LIN {X 0,Y 574.087,Z 352.568,A -85,B 0,C 180,E1 -2236.257,E2 -2236.257} C_VEL
LIN {X 0,Y 573.893,Z 454.984,A -85,B 0,C 180,E1 -2237.558,E2 -2237.558} C_VEL
LIN {X 0,Y 573.782,Z 468.244,A -85,B 0,C 180,E1 -2237.87,E2 -2237.87} C_VEL
LIN {X 0,Y 573.666,Z 481.513,A -85,B 0,C 180,E1 -2238.339,E2 -2238.339} C_VEL
LIN {X 0,Y 573.595,Z 492.64,A -85,B 0,C 180,E1 -2238.874,E2 -2238.874} C_VEL
LIN {X 0,Y 573.43,Z 504.211,A -85,B 0,C 180,E1 -2239.586,E2 -2239.586} C_VEL
LIN {X 0,Y 573.326,Z 514.578,A -85,B 0,C 180,E1 -2240.386,E2 -2240.386} C_VEL
LIN {X 0,Y 573.238,Z 523.076,A -85,B 0,C 180,E1 -2241.185,E2 -2241.185} C_VEL
LIN {X 0,Y 573.16,Z 530.966,A -85,B 0,C 180,E1 -2242.072,E2 -2242.072} C_VEL
LIN {X 0,Y 573.078,Z 538.898,A -85,B 0,C 180,E1 -2243.177,E2 -2243.177} C_VEL
LIN {X 0,Y 573.07,Z 545.683,A -85,B 0,C 180,E1 -2244.37,E2 -2244.37} C_VEL
LIN {X 0,Y 573.028,Z 550.375,A -85,B 0,C 180,E1 -2245.428,E2 -2245.428} C_VEL
LIN {X 0,Y 573.023,Z 553.959,A -85,B 0,C 180,E1 -2246.485,E2 -2246.485} C_VEL
LIN {X 0,Y 572.959,Z 555.81,A -85,B 0,C 180,E1 -2247.188,E2 -2247.188} C_VEL
LIN {X 0,Y 572.946,Z 558.186,A -85,B 0,C 180,E1 -2248.595,E2 -2248.595} C_VEL
LIN {X 0,Y 572.938,Z 559,A -85,B 0,C 180,E1 -2250.001,E2 -2250.001} C_VEL
LIN {X 0,Y 572.946,Z 558.186,A -85,B 0,C 180,E1 -2251.406,E2 -2251.406} C_VEL
LIN {X 0,Y 572.937,Z 557.198,A -85,B 0,C 180,E1 -2252.11,E2 -2252.11} C_VEL
LIN {X 0,Y 572.959,Z 555.808,A -85,B 0,C 180,E1 -2252.813,E2 -2252.813} C_VEL
LIN {X 0,Y 573.014,Z 552.894,A -85,B 0,C 180,E1 -2253.869,E2 -2253.869} C_VEL
LIN {X 0,Y 572.963,Z 548.946,A -85,B 0,C 180,E1 -2254.926,E2 -2254.926} C_VEL
LIN {X 0,Y 573.067,Z 542.873,A -85,B 0,C 180,E1 -2256.161,E2 -2256.161} C_VEL
LIN {X 0,Y 573.12,Z 536.233,A -85,B 0,C 180,E1 -2257.221,E2 -2257.221} C_VEL
LIN {X 0,Y 573.192,Z 527.986,A -85,B 0,C 180,E1 -2258.284,E2 -2258.284} C_VEL
LIN {X 0,Y 573.312,Z 517.586,A -85,B 0,C 180,E1 -2259.348,E2 -2259.348} C_VEL
LIN {X 0,Y 573.427,Z 507.917,A -85,B 0,C 180,E1 -2260.148,E2 -2260.148} C_VEL
LIN {X 0,Y 573.552,Z 497.347,A -85,B 0,C 180,E1 -2260.858,E2 -2260.858} C_VEL
LIN {X 0,Y 573.654,Z 486.27,A -85,B 0,C 180,E1 -2261.448,E2 -2261.448} C_VEL
LIN {X 0,Y 573.76,Z 473.155,A -85,B 0,C 180,E1 -2261.975,E2 -2261.975} C_VEL
LIN {X 0,Y 573.831,Z 460.495,A -85,B 0,C 180,E1 -2262.332,E2 -2262.332} C_VEL
LIN {X 0,Y 573.897,Z 447.265,A -85,B 0,C 180,E1 -2262.555,E2 -2262.555} C_VEL
LIN {X 0,Y 573.953,Z 350.676,A -85,B 0,C 180,E1 -2263.77,E2 -2263.77} C_VEL
LIN {X 0,Y 573.386,Z 346.788,A -85,B 0,C 180,E1 -2263.851,E2 -2263.851} C_VEL
LIN {X 0,Y 573.57,Z 325.022,A -85,B 0,C 180,E1 -2266.994,E2 -2266.994} C_VEL
LIN {X 0,Y 573.803,Z 304.129,A -85,B 0,C 180,E1 -2270.057,E2 -2270.057} C_VEL
LIN {X 0,Y 573.969,Z 288.92,A -85,B 0,C 180,E1 -2272.308,E2 -2272.308} C_VEL
LIN {X 0,Y 573.237,Z 284.083,A -85,B 0,C 180,E1 -2273.076,E2 -2273.076} C_VEL
LIN {X 0,Y 573.243,Z 284.082,A -85,B 0,C 180,E1 -2275.411,E2 -2275.411} C_VEL
LIN {X 0,Y 573.25,Z 284.078,A -85,B 0,C 180,E1 -2278.028,E2 -2278.028} C_VEL
LIN {X 0,Y 573.222,Z 284.075,A -85,B 0,C 180,E1 -2280.994,E2 -2280.994} C_VEL
LIN {X 0,Y 573.267,Z 284.073,A -85,B 0,C 180,E1 -2283.524,E2 -2283.524} C_VEL
LIN {X 0,Y 573.193,Z 284.09,A -85,B 0,C 180,E1 -2286.054,E2 -2286.054} C_VEL
LIN {X 0,Y 573.24,Z 284.075,A -85,B 0,C 180,E1 -2288.702,E2 -2288.702} C_VEL
LIN {X 0,Y 573.219,Z 284.077,A -85,B 0,C 180,E1 -2291.591,E2 -2291.591} C_VEL
LIN {X 0,Y 573.221,Z 284.086,A -85,B 0,C 180,E1 -2294.335,E2 -2294.335} C_VEL
LIN {X 0,Y 573.236,Z 284.073,A -85,B 0,C 180,E1 -2297.36,E2 -2297.36} C_VEL
LIN {X 0,Y 573.24,Z 284.08,A -85,B 0,C 180,E1 -2300.392,E2 -2300.392} C_VEL
LIN {X 0,Y 573.234,Z 284.078,A -85,B 0,C 180,E1 -2303.076,E2 -2303.076} C_VEL
LIN {X 0,Y 573.265,Z 284.07,A -85,B 0,C 180,E1 -2305.671,E2 -2305.671} C_VEL
LIN {X 0,Y 573.238,Z 284.074,A -85,B 0,C 180,E1 -2308.184,E2 -2308.184} C_VEL
LIN {X 0,Y 573.261,Z 284.075,A -85,B 0,C 180,E1 -2310.634,E2 -2310.634} C_VEL
LIN {X 0,Y 573.215,Z 284.086,A -85,B 0,C 180,E1 -2313.022,E2 -2313.022} C_VEL
LIN {X 0,Y 573.221,Z 284.083,A -85,B 0,C 180,E1 -2315.363,E2 -2315.363} C_VEL
LIN {X 0,Y 573.228,Z 284.078,A -85,B 0,C 180,E1 -2317.662,E2 -2317.662} C_VEL
LIN {X 0,Y 573.241,Z 284.075,A -85,B 0,C 180,E1 -2319.923,E2 -2319.923} C_VEL
LIN {X 0,Y 573.263,Z 284.073,A -85,B 0,C 180,E1 -2322.99,E2 -2322.99} C_VEL
LIN {X 0,Y 573.266,Z 284.076,A -85,B 0,C 180,E1 -2325.807,E2 -2325.807} C_VEL
LIN {X 0,Y 573.267,Z 284.069,A -85,B 0,C 180,E1 -2328.745,E2 -2328.745} C_VEL
LIN {X 0,Y 573.247,Z 284.079,A -85,B 0,C 180,E1 -2331.54,E2 -2331.54} C_VEL
LIN {X 0,Y 573.241,Z 284.08,A -85,B 0,C 180,E1 -2333.665,E2 -2333.665} C_VEL
LIN {X 0,Y 573.227,Z 284.083,A -85,B 0,C 180,E1 -2335.781,E2 -2335.781} C_VEL
LIN {X 0,Y 573.316,Z 284.072,A -85,B 0,C 180,E1 -2337.892,E2 -2337.892} C_VEL
LIN {X 0,Y 573.319,Z 284.065,A -85,B 0,C 180,E1 -2340.702,E2 -2340.702} C_VEL
LIN {X 0,Y 573.293,Z 284.068,A -85,B 0,C 180,E1 -2342.811,E2 -2342.811} C_VEL
LIN {X 0,Y 573.279,Z 284.069,A -85,B 0,C 180,E1 -2345.628,E2 -2345.628} C_VEL
LIN {X 0,Y 573.282,Z 284.079,A -85,B 0,C 180,E1 -2348.459,E2 -2348.459} C_VEL
LIN {X 0,Y 573.275,Z 284.069,A -85,B 0,C 180,E1 -2351.312,E2 -2351.312} C_VEL
LIN {X 0,Y 573.283,Z 284.074,A -85,B 0,C 180,E1 -2354.424,E2 -2354.424} C_VEL
LIN {X 0,Y 573.26,Z 284.075,A -85,B 0,C 180,E1 -2357.111,E2 -2357.111} C_VEL
LIN {X 0,Y 573.241,Z 284.073,A -85,B 0,C 180,E1 -2360.077,E2 -2360.077} C_VEL
LIN {X 0,Y 573.232,Z 284.075,A -85,B 0,C 180,E1 -2362.338,E2 -2362.338} C_VEL
LIN {X 0,Y 573.244,Z 284.073,A -85,B 0,C 180,E1 -2364.377,E2 -2364.377} C_VEL
LIN {X 0,Y 572.618,Z 284.16,A -85,B 0,C 180,E1 -2364.963,E2 -2364.963} C_VEL
LIN {X 0,Y 569.762,Z 284.519,A -85,B 0,C 180,E1 -2365.914,E2 -2365.914} C_VEL
LIN {X 0,Y 567.319,Z 284.824,A -85,B 0,C 180,E1 -2366.68,E2 -2366.68} C_VEL
LIN {X 0,Y 566.261,Z 284.951,A -85,B 0,C 180,E1 -2367.271,E2 -2367.271} C_VEL
LIN {X 0,Y 566.172,Z 284.959,A -85,B 0,C 180,E1 -2367.471,E2 -2367.471} C_VEL
LIN {X 0,Y 566.197,Z 284.953,A -85,B 0,C 180,E1 -2369.769,E2 -2369.769} C_VEL
LIN {X 0,Y 566.202,Z 284.949,A -85,B 0,C 180,E1 -2372.429,E2 -2372.429} C_VEL
LIN {X 0,Y 566.185,Z 284.955,A -85,B 0,C 180,E1 -2374.99,E2 -2374.99} C_VEL
LIN {X 0,Y 566.193,Z 284.96,A -85,B 0,C 180,E1 -2377.461,E2 -2377.461} C_VEL
LIN {X 0,Y 566.21,Z 284.951,A -85,B 0,C 180,E1 -2380.199,E2 -2380.199} C_VEL
LIN {X 0,Y 566.194,Z 284.951,A -85,B 0,C 180,E1 -2383.055,E2 -2383.055} C_VEL
LIN {X 0,Y 566.195,Z 284.958,A -85,B 0,C 180,E1 -2386.049,E2 -2386.049} C_VEL
LIN {X 0,Y 566.205,Z 284.95,A -85,B 0,C 180,E1 -2389.214,E2 -2389.214} C_VEL
LIN {X 0,Y 566.179,Z 284.956,A -85,B 0,C 180,E1 -2391.636,E2 -2391.636} C_VEL
LIN {X 0,Y 566.152,Z 284.965,A -85,B 0,C 180,E1 -2394.307,E2 -2394.307} C_VEL
LIN {X 0,Y 566.212,Z 284.95,A -85,B 0,C 180,E1 -2396.897,E2 -2396.897} C_VEL
LIN {X 0,Y 566.179,Z 284.952,A -85,B 0,C 180,E1 -2399.407,E2 -2399.407} C_VEL
LIN {X 0,Y 566.192,Z 284.952,A -85,B 0,C 180,E1 -2401.856,E2 -2401.856} C_VEL
LIN {X 0,Y 566.195,Z 284.956,A -85,B 0,C 180,E1 -2404.25,E2 -2404.25} C_VEL
LIN {X 0,Y 566.167,Z 284.964,A -85,B 0,C 180,E1 -2406.72,E2 -2406.72} C_VEL
LIN {X 0,Y 566.203,Z 284.949,A -85,B 0,C 180,E1 -2409.662,E2 -2409.662} C_VEL
LIN {X 0,Y 566.181,Z 284.952,A -85,B 0,C 180,E1 -2411.921,E2 -2411.921} C_VEL
LIN {X 0,Y 566.19,Z 284.951,A -85,B 0,C 180,E1 -2414.152,E2 -2414.152} C_VEL
LIN {X 0,Y 566.182,Z 284.953,A -85,B 0,C 180,E1 -2416.358,E2 -2416.358} C_VEL
LIN {X 0,Y 566.235,Z 284.949,A -85,B 0,C 180,E1 -2418.676,E2 -2418.676} C_VEL
LIN {X 0,Y 566.195,Z 284.96,A -85,B 0,C 180,E1 -2421.433,E2 -2421.433} C_VEL
LIN {X 0,Y 566.273,Z 285.018,A -85,B 0,C 180,E1 -2424.19,E2 -2424.19} C_VEL
LIN {X 0,Y 566.485,Z 289.646,A -85,B 0,C 180,E1 -2425.017,E2 -2425.017} C_VEL
LIN {X 0,Y 566.399,Z 303.708,A -85,B 0,C 180,E1 -2427.51,E2 -2427.51} C_VEL
LIN {X 0,Y 566.29,Z 318.14,A -85,B 0,C 180,E1 -2430.044,E2 -2430.044} C_VEL
LIN {X 0,Y 567.193,Z 324.333,A -85,B 0,C 180,E1 -2430.155,E2 -2430.155} C_VEL
LIN {X 0,Y 566.973,Z 424.618,A -85,B 0,C 180,E1 -2431.442,E2 -2431.442} C_VEL
LIN {X 0,Y 566.822,Z 437.137,A -85,B 0,C 180,E1 -2431.731,E2 -2431.731} C_VEL
LIN {X 0,Y 566.703,Z 449.964,A -85,B 0,C 180,E1 -2432.176,E2 -2432.176} C_VEL
LIN {X 0,Y 566.6,Z 462.185,A -85,B 0,C 180,E1 -2432.754,E2 -2432.754} C_VEL
LIN {X 0,Y 566.444,Z 473.726,A -85,B 0,C 180,E1 -2433.467,E2 -2433.467} C_VEL
LIN {X 0,Y 566.293,Z 484.13,A -85,B 0,C 180,E1 -2434.27,E2 -2434.27} C_VEL
LIN {X 0,Y 566.188,Z 493.498,A -85,B 0,C 180,E1 -2435.163,E2 -2435.163} C_VEL
LIN {X 0,Y 566.112,Z 501.276,A -85,B 0,C 180,E1 -2436.057,E2 -2436.057} C_VEL
LIN {X 0,Y 566.01,Z 508.874,A -85,B 0,C 180,E1 -2437.132,E2 -2437.132} C_VEL
LIN {X 0,Y 565.977,Z 514.998,A -85,B 0,C 180,E1 -2438.209,E2 -2438.209} C_VEL
LIN {X 0,Y 565.893,Z 519.877,A -85,B 0,C 180,E1 -2439.29,E2 -2439.29} C_VEL
LIN {X 0,Y 565.902,Z 523.628,A -85,B 0,C 180,E1 -2440.374,E2 -2440.374} C_VEL
LIN {X 0,Y 565.87,Z 526.355,A -85,B 0,C 180,E1 -2441.461,E2 -2441.461} C_VEL
LIN {X 0,Y 565.864,Z 527.635,A -85,B 0,C 180,E1 -2442.188,E2 -2442.188} C_VEL
LIN {X 0,Y 565.843,Z 528.504,A -85,B 0,C 180,E1 -2442.918,E2 -2442.918} C_VEL
LIN {X 0,Y 565.861,Z 528.919,A -85,B 0,C 180,E1 -2443.649,E2 -2443.649} C_VEL
LIN {X 0,Y 565.874,Z 528.932,A -85,B 0,C 180,E1 -2444.382,E2 -2444.382} C_VEL
LIN {X 0,Y 565.809,Z 528.542,A -85,B 0,C 180,E1 -2445.119,E2 -2445.119} C_VEL
LIN {X 0,Y 565.828,Z 527.702,A -85,B 0,C 180,E1 -2445.857,E2 -2445.857} C_VEL
LIN {X 0,Y 565.855,Z 525.567,A -85,B 0,C 180,E1 -2446.991,E2 -2446.991} C_VEL
LIN {X 0,Y 565.911,Z 522.48,A -85,B 0,C 180,E1 -2448.087,E2 -2448.087} C_VEL
LIN {X 0,Y 565.95,Z 517.743,A -85,B 0,C 180,E1 -2449.305,E2 -2449.305} C_VEL
LIN {X 0,Y 565.993,Z 511.457,A -85,B 0,C 180,E1 -2450.534,E2 -2450.534} C_VEL
LIN {X 0,Y 566.062,Z 504.858,A -85,B 0,C 180,E1 -2451.556,E2 -2451.556} C_VEL
LIN {X 0,Y 566.141,Z 496.229,A -85,B 0,C 180,E1 -2452.632,E2 -2452.632} C_VEL
LIN {X 0,Y 566.289,Z 486.697,A -85,B 0,C 180,E1 -2453.592,E2 -2453.592} C_VEL
LIN {X 0,Y 566.364,Z 477.313,A -85,B 0,C 180,E1 -2454.367,E2 -2454.367} C_VEL
LIN {X 0,Y 566.527,Z 466.377,A -85,B 0,C 180,E1 -2455.097,E2 -2455.097} C_VEL
LIN {X 0,Y 566.675,Z 454.313,A -85,B 0,C 180,E1 -2455.726,E2 -2455.726} C_VEL
LIN {X 0,Y 566.782,Z 441.869,A -85,B 0,C 180,E1 -2456.214,E2 -2456.214} C_VEL
LIN {X 0,Y 566.893,Z 429.518,A -85,B 0,C 180,E1 -2456.552,E2 -2456.552} C_VEL
LIN {X 0,Y 566.993,Z 413.576,A -85,B 0,C 180,E1 -2456.802,E2 -2456.802} C_VEL
LIN {X 0,Y 567.037,Z 322.815,A -85,B 0,C 180,E1 -2457.959,E2 -2457.959} C_VEL
LIN {X 0,Y 566.264,Z 318.046,A -85,B 0,C 180,E1 -2458.063,E2 -2458.063} C_VEL
LIN {X 0,Y 566.443,Z 302.182,A -85,B 0,C 180,E1 -2460.848,E2 -2460.848} C_VEL
LIN {X 0,Y 566.536,Z 287.643,A -85,B 0,C 180,E1 -2463.407,E2 -2463.407} C_VEL
LIN {X 0,Y 566.189,Z 284.958,A -85,B 0,C 180,E1 -2463.89,E2 -2463.89} C_VEL
LIN {X 0,Y 566.192,Z 284.959,A -85,B 0,C 180,E1 -2466.569,E2 -2466.569} C_VEL
LIN {X 0,Y 566.204,Z 284.951,A -85,B 0,C 180,E1 -2469.685,E2 -2469.685} C_VEL
LIN {X 0,Y 566.186,Z 284.961,A -85,B 0,C 180,E1 -2472.916,E2 -2472.916} C_VEL
LIN {X 0,Y 566.15,Z 284.957,A -85,B 0,C 180,E1 -2476.053,E2 -2476.053} C_VEL
LIN {X 0,Y 566.157,Z 284.961,A -85,B 0,C 180,E1 -2478.859,E2 -2478.859} C_VEL
LIN {X 0,Y 566.195,Z 284.959,A -85,B 0,C 180,E1 -2481.442,E2 -2481.442} C_VEL
LIN {X 0,Y 566.152,Z 284.956,A -85,B 0,C 180,E1 -2484.307,E2 -2484.307} C_VEL
LIN {X 0,Y 566.188,Z 284.951,A -85,B 0,C 180,E1 -2486.896,E2 -2486.896} C_VEL
LIN {X 0,Y 566.157,Z 284.965,A -85,B 0,C 180,E1 -2489.406,E2 -2489.406} C_VEL
LIN {X 0,Y 566.178,Z 284.959,A -85,B 0,C 180,E1 -2491.856,E2 -2491.856} C_VEL
LIN {X 0,Y 566.165,Z 284.956,A -85,B 0,C 180,E1 -2494.249,E2 -2494.249} C_VEL
LIN {X 0,Y 566.156,Z 284.956,A -85,B 0,C 180,E1 -2496.72,E2 -2496.72} C_VEL
LIN {X 0,Y 566.19,Z 284.959,A -85,B 0,C 180,E1 -2499.662,E2 -2499.662} C_VEL
LIN {X 0,Y 566.154,Z 284.965,A -85,B 0,C 180,E1 -2501.92,E2 -2501.92} C_VEL
LIN {X 0,Y 566.168,Z 284.954,A -85,B 0,C 180,E1 -2504.89,E2 -2504.89} C_VEL
LIN {X 0,Y 566.165,Z 284.959,A -85,B 0,C 180,E1 -2507.818,E2 -2507.818} C_VEL
LIN {X 0,Y 566.147,Z 284.965,A -85,B 0,C 180,E1 -2509.992,E2 -2509.992} C_VEL
LIN {X 0,Y 566.171,Z 284.955,A -85,B 0,C 180,E1 -2512.87,E2 -2512.87} C_VEL
LIN {X 0,Y 566.232,Z 284.947,A -85,B 0,C 180,E1 -2515.016,E2 -2515.016} C_VEL
LIN {X 0,Y 566.246,Z 284.946,A -85,B 0,C 180,E1 -2517.866,E2 -2517.866} C_VEL
LIN {X 0,Y 566.287,Z 284.945,A -85,B 0,C 180,E1 -2520.711,E2 -2520.711} C_VEL
LIN {X 0,Y 566.248,Z 284.949,A -85,B 0,C 180,E1 -2522.846,E2 -2522.846} C_VEL
LIN {X 0,Y 566.216,Z 284.948,A -85,B 0,C 180,E1 -2525.699,E2 -2525.699} C_VEL
LIN {X 0,Y 566.171,Z 284.952,A -85,B 0,C 180,E1 -2527.848,E2 -2527.848} C_VEL
LIN {X 0,Y 566.209,Z 284.959,A -85,B 0,C 180,E1 -2530.73,E2 -2530.73} C_VEL
LIN {X 0,Y 566.156,Z 284.954,A -85,B 0,C 180,E1 -2533.642,E2 -2533.642} C_VEL
LIN {X 0,Y 566.166,Z 284.959,A -85,B 0,C 180,E1 -2536.589,E2 -2536.589} C_VEL
LIN {X 0,Y 566.189,Z 284.953,A -85,B 0,C 180,E1 -2539.582,E2 -2539.582} C_VEL
LIN {X 0,Y 566.176,Z 284.953,A -85,B 0,C 180,E1 -2541.863,E2 -2541.863} C_VEL
LIN {X 0,Y 566.17,Z 284.961,A -85,B 0,C 180,E1 -2545.022,E2 -2545.022} C_VEL
LIN {X 0,Y 566.166,Z 284.963,A -85,B 0,C 180,E1 -2547.342,E2 -2547.342} C_VEL
LIN {X 0,Y 566.162,Z 284.959,A -85,B 0,C 180,E1 -2549.771,E2 -2549.771} C_VEL
LIN {X 0,Y 566.192,Z 284.951,A -85,B 0,C 180,E1 -2552.43,E2 -2552.43} C_VEL
LIN {X 0,Y 566.169,Z 284.957,A -85,B 0,C 180,E1 -2554.989,E2 -2554.989} C_VEL
LIN {X 0,Y 566.185,Z 284.961,A -85,B 0,C 180,E1 -2557.462,E2 -2557.462} C_VEL
LIN {X 0,Y 566.2,Z 284.953,A -85,B 0,C 180,E1 -2560.2,E2 -2560.2} C_VEL
LIN {X 0,Y 566.189,Z 284.951,A -85,B 0,C 180,E1 -2563.056,E2 -2563.056} C_VEL
LIN {X 0,Y 566.188,Z 284.96,A -85,B 0,C 180,E1 -2566.05,E2 -2566.05} C_VEL
LIN {X 0,Y 566.199,Z 284.952,A -85,B 0,C 180,E1 -2569.216,E2 -2569.216} C_VEL
LIN {X 0,Y 566.177,Z 284.958,A -85,B 0,C 180,E1 -2571.637,E2 -2571.637} C_VEL
LIN {X 0,Y 566.146,Z 284.964,A -85,B 0,C 180,E1 -2574.308,E2 -2574.308} C_VEL
LIN {X 0,Y 566.217,Z 284.95,A -85,B 0,C 180,E1 -2576.899,E2 -2576.899} C_VEL
LIN {X 0,Y 566.173,Z 284.955,A -85,B 0,C 180,E1 -2579.408,E2 -2579.408} C_VEL
LIN {X 0,Y 566.193,Z 284.956,A -85,B 0,C 180,E1 -2581.857,E2 -2581.857} C_VEL
LIN {X 0,Y 566.203,Z 284.961,A -85,B 0,C 180,E1 -2584.251,E2 -2584.251} C_VEL
LIN {X 0,Y 566.193,Z 285.017,A -85,B 0,C 180,E1 -2586.825,E2 -2586.825} C_VEL
LIN {X 0,Y 566.991,Z 289.95,A -85,B 0,C 180,E1 -2587.596,E2 -2587.596} C_VEL
LIN {X 0,Y 566.811,Z 307.864,A -85,B 0,C 180,E1 -2590.253,E2 -2590.253} C_VEL
LIN {X 0,Y 566.587,Z 325.666,A -85,B 0,C 180,E1 -2592.885,E2 -2592.885} C_VEL
LIN {X 0,Y 566.401,Z 346.64,A -85,B 0,C 180,E1 -2595.953,E2 -2595.953} C_VEL
LIN {X 0,Y 566.42,Z 347.202,A -85,B 0,C 180,E1 -2595.999,E2 -2595.999} C_VEL
LIN {X 0,Y 567.19,Z 353.35,A -85,B 0,C 180,E1 -2596.097,E2 -2596.097} C_VEL
LIN {X 0,Y 566.981,Z 454.984,A -85,B 0,C 180,E1 -2597.404,E2 -2597.404} C_VEL
LIN {X 0,Y 566.852,Z 468.243,A -85,B 0,C 180,E1 -2597.72,E2 -2597.72} C_VEL
LIN {X 0,Y 566.712,Z 481.513,A -85,B 0,C 180,E1 -2598.194,E2 -2598.194} C_VEL
LIN {X 0,Y 566.62,Z 493.17,A -85,B 0,C 180,E1 -2598.766,E2 -2598.766} C_VEL
LIN {X 0,Y 566.444,Z 504.209,A -85,B 0,C 180,E1 -2599.456,E2 -2599.456} C_VEL
LIN {X 0,Y 566.317,Z 514.593,A -85,B 0,C 180,E1 -2600.266,E2 -2600.266} C_VEL
LIN {X 0,Y 566.21,Z 523.09,A -85,B 0,C 180,E1 -2601.075,E2 -2601.075} C_VEL
LIN {X 0,Y 566.11,Z 530.966,A -85,B 0,C 180,E1 -2601.972,E2 -2601.972} C_VEL
LIN {X 0,Y 566.004,Z 538.626,A -85,B 0,C 180,E1 -2603.047,E2 -2603.047} C_VEL
LIN {X 0,Y 566.003,Z 545.683,A -85,B 0,C 180,E1 -2604.3,E2 -2604.3} C_VEL
LIN {X 0,Y 565.933,Z 550.375,A -85,B 0,C 180,E1 -2605.371,E2 -2605.371} C_VEL
LIN {X 0,Y 565.927,Z 553.96,A -85,B 0,C 180,E1 -2606.441,E2 -2606.441} C_VEL
LIN {X 0,Y 565.878,Z 555.809,A -85,B 0,C 180,E1 -2607.153,E2 -2607.153} C_VEL
LIN {X 0,Y 565.846,Z 558.185,A -85,B 0,C 180,E1 -2608.577,E2 -2608.577} C_VEL
LIN {X 0,Y 565.839,Z 559,A -85,B 0,C 180,E1 -2610.001,E2 -2610.001} C_VEL
LIN {X 0,Y 565.846,Z 558.185,A -85,B 0,C 180,E1 -2611.424,E2 -2611.424} C_VEL
LIN {X 0,Y 565.878,Z 555.809,A -85,B 0,C 180,E1 -2612.848,E2 -2612.848} C_VEL
LIN {X 0,Y 565.926,Z 552.894,A -85,B 0,C 180,E1 -2613.917,E2 -2613.917} C_VEL
LIN {X 0,Y 565.878,Z 548.946,A -85,B 0,C 180,E1 -2614.988,E2 -2614.988} C_VEL
LIN {X 0,Y 565.994,Z 542.873,A -85,B 0,C 180,E1 -2616.238,E2 -2616.238} C_VEL
LIN {X 0,Y 566.052,Z 536.233,A -85,B 0,C 180,E1 -2617.312,E2 -2617.312} C_VEL
LIN {X 0,Y 566.141,Z 527.986,A -85,B 0,C 180,E1 -2618.388,E2 -2618.388} C_VEL
LIN {X 0,Y 566.274,Z 519.533,A -85,B 0,C 180,E1 -2619.285,E2 -2619.285} C_VEL
LIN {X 0,Y 566.413,Z 509.088,A -85,B 0,C 180,E1 -2620.185,E2 -2620.185} C_VEL
LIN {X 0,Y 566.571,Z 497.663,A -85,B 0,C 180,E1 -2620.973,E2 -2620.973} C_VEL
LIN {X 0,Y 566.696,Z 485.874,A -85,B 0,C 180,E1 -2621.609,E2 -2621.609} C_VEL
LIN {X 0,Y 566.814,Z 473.153,A -85,B 0,C 180,E1 -2622.123,E2 -2622.123} C_VEL
LIN {X 0,Y 566.894,Z 460.494,A -85,B 0,C 180,E1 -2622.485,E2 -2622.485} C_VEL
LIN {X 0,Y 566.979,Z 447.265,A -85,B 0,C 180,E1 -2622.711,E2 -2622.711} C_VEL
LIN {X 0,Y 567.051,Z 351.346,A -85,B 0,C 180,E1 -2623.932,E2 -2623.932} C_VEL
LIN {X 0,Y 566.384,Z 346.788,A -85,B 0,C 180,E1 -2624.026,E2 -2624.026} C_VEL
LIN {X 0,Y 566.591,Z 325.657,A -85,B 0,C 180,E1 -2627.116,E2 -2627.116} C_VEL
LIN {X 0,Y 566.861,Z 305.32,A -85,B 0,C 180,E1 -2630.124,E2 -2630.124} C_VEL
LIN {X 0,Y 567.017,Z 290.018,A -85,B 0,C 180,E1 -2632.405,E2 -2632.405} C_VEL
LIN {X 0,Y 566.179,Z 284.963,A -85,B 0,C 180,E1 -2633.201,E2 -2633.201} C_VEL
LIN {X 0,Y 566.207,Z 284.96,A -85,B 0,C 180,E1 -2635.75,E2 -2635.75} C_VEL
LIN {X 0,Y 566.208,Z 284.953,A -85,B 0,C 180,E1 -2638.202,E2 -2638.202} C_VEL
LIN {X 0,Y 566.189,Z 284.952,A -85,B 0,C 180,E1 -2641.075,E2 -2641.075} C_VEL
LIN {X 0,Y 566.215,Z 284.955,A -85,B 0,C 180,E1 -2643.734,E2 -2643.734} C_VEL
LIN {X 0,Y 566.184,Z 284.954,A -85,B 0,C 180,E1 -2646.572,E2 -2646.572} C_VEL
LIN {X 0,Y 566.216,Z 284.951,A -85,B 0,C 180,E1 -2649.685,E2 -2649.685} C_VEL
LIN {X 0,Y 566.186,Z 284.959,A -85,B 0,C 180,E1 -2652.09,E2 -2652.09} C_VEL
LIN {X 0,Y 566.168,Z 284.955,A -85,B 0,C 180,E1 -2655.037,E2 -2655.037} C_VEL
LIN {X 0,Y 566.19,Z 284.953,A -85,B 0,C 180,E1 -2657.91,E2 -2657.91} C_VEL
LIN {X 0,Y 566.214,Z 284.957,A -85,B 0,C 180,E1 -2660.726,E2 -2660.726} C_VEL
LIN {X 0,Y 566.185,Z 284.953,A -85,B 0,C 180,E1 -2663.429,E2 -2663.429} C_VEL
LIN {X 0,Y 566.215,Z 284.95,A -85,B 0,C 180,E1 -2666.266,E2 -2666.266} C_VEL
LIN {X 0,Y 566.188,Z 284.963,A -85,B 0,C 180,E1 -2668.925,E2 -2668.925} C_VEL
LIN {X 0,Y 566.194,Z 284.951,A -85,B 0,C 180,E1 -2671.856,E2 -2671.856} C_VEL
LIN {X 0,Y 566.196,Z 284.95,A -85,B 0,C 180,E1 -2674.25,E2 -2674.25} C_VEL
LIN {X 0,Y 566.176,Z 284.961,A -85,B 0,C 180,E1 -2677.368,E2 -2677.368} C_VEL
LIN {X 0,Y 566.208,Z 284.954,A -85,B 0,C 180,E1 -2679.662,E2 -2679.662} C_VEL
LIN {X 0,Y 566.2,Z 284.95,A -85,B 0,C 180,E1 -2682.668,E2 -2682.668} C_VEL
LIN {X 0,Y 566.23,Z 284.956,A -85,B 0,C 180,E1 -2685.627,E2 -2685.627} C_VEL
LIN {X 0,Y 566.238,Z 284.945,A -85,B 0,C 180,E1 -2688.675,E2 -2688.675} C_VEL
LIN {X 0,Y 566.2,Z 284.955,A -85,B 0,C 180,E1 -2691.434,E2 -2691.434} C_VEL
LIN {X 0,Y 566.205,Z 284.955,A -85,B 0,C 180,E1 -2693.586,E2 -2693.586} C_VEL
LIN {X 0,Y 566.185,Z 284.959,A -85,B 0,C 180,E1 -2695.729,E2 -2695.729} C_VEL
LIN {X 0,Y 566.286,Z 284.947,A -85,B 0,C 180,E1 -2697.866,E2 -2697.866} C_VEL
LIN {X 0,Y 566.291,Z 284.94,A -85,B 0,C 180,E1 -2700.711,E2 -2700.711} C_VEL
LIN {X 0,Y 566.261,Z 284.944,A -85,B 0,C 180,E1 -2702.845,E2 -2702.845} C_VEL
LIN {X 0,Y 566.248,Z 284.945,A -85,B 0,C 180,E1 -2705.698,E2 -2705.698} C_VEL
LIN {X 0,Y 566.226,Z 284.955,A -85,B 0,C 180,E1 -2708.566,E2 -2708.566} C_VEL
LIN {X 0,Y 566.245,Z 284.944,A -85,B 0,C 180,E1 -2711.454,E2 -2711.454} C_VEL
LIN {X 0,Y 566.236,Z 284.953,A -85,B 0,C 180,E1 -2714.506,E2 -2714.506} C_VEL
LIN {X 0,Y 566.198,Z 284.952,A -85,B 0,C 180,E1 -2717.332,E2 -2717.332} C_VEL
LIN {X 0,Y 566.208,Z 284.951,A -85,B 0,C 180,E1 -2720.337,E2 -2720.337} C_VEL
LIN {X 0,Y 566.168,Z 284.96,A -85,B 0,C 180,E1 -2723.28,E2 -2723.28} C_VEL
LIN {X 0,Y 566.206,Z 284.95,A -85,B 0,C 180,E1 -2725.749,E2 -2725.749} C_VEL
LIN {X 0,Y 566.172,Z 284.959,A -85,B 0,C 180,E1 -2727.471,E2 -2727.471} C_VEL
LIN {X 0,Y 565.499,Z 285.04,A -85,B 0,C 180,E1 -2728.065,E2 -2728.065} C_VEL
LIN {X 0,Y 562.644,Z 285.4,A -85,B 0,C 180,E1 -2729.029,E2 -2729.029} C_VEL
LIN {X 0,Y 560.241,Z 285.695,A -85,B 0,C 180,E1 -2729.805,E2 -2729.805} C_VEL
LIN {X 0,Y 559.215,Z 285.82,A -85,B 0,C 180,E1 -2730.404,E2 -2730.404} C_VEL
LIN {X 0,Y 559.135,Z 285.831,A -85,B 0,C 180,E1 -2730.607,E2 -2730.607} C_VEL
LIN {X 0,Y 559.153,Z 285.829,A -85,B 0,C 180,E1 -2732.715,E2 -2732.715} C_VEL
LIN {X 0,Y 559.127,Z 285.839,A -85,B 0,C 180,E1 -2735.324,E2 -2735.324} C_VEL
LIN {X 0,Y 559.131,Z 285.834,A -85,B 0,C 180,E1 -2738.018,E2 -2738.018} C_VEL
LIN {X 0,Y 559.156,Z 285.827,A -85,B 0,C 180,E1 -2740.812,E2 -2740.812} C_VEL
LIN {X 0,Y 559.138,Z 285.84,A -85,B 0,C 180,E1 -2743.734,E2 -2743.734} C_VEL
LIN {X 0,Y 559.143,Z 285.829,A -85,B 0,C 180,E1 -2746.804,E2 -2746.804} C_VEL
LIN {X 0,Y 559.156,Z 285.828,A -85,B 0,C 180,E1 -2749.187,E2 -2749.187} C_VEL
LIN {X 0,Y 559.127,Z 285.84,A -85,B 0,C 180,E1 -2751.981,E2 -2751.981} C_VEL
LIN {X 0,Y 559.13,Z 285.833,A -85,B 0,C 180,E1 -2754.787,E2 -2754.787} C_VEL
LIN {X 0,Y 559.156,Z 285.827,A -85,B 0,C 180,E1 -2757.364,E2 -2757.364} C_VEL
LIN {X 0,Y 559.148,Z 285.834,A -85,B 0,C 180,E1 -2760.143,E2 -2760.143} C_VEL
LIN {X 0,Y 559.16,Z 285.828,A -85,B 0,C 180,E1 -2763.175,E2 -2763.175} C_VEL
LIN {X 0,Y 559.125,Z 285.831,A -85,B 0,C 180,E1 -2765.493,E2 -2765.493} C_VEL
LIN {X 0,Y 559.172,Z 285.834,A -85,B 0,C 180,E1 -2768.623,E2 -2768.623} C_VEL
LIN {X 0,Y 559.159,Z 285.836,A -85,B 0,C 180,E1 -2770.925,E2 -2770.925} C_VEL
LIN {X 0,Y 559.154,Z 285.827,A -85,B 0,C 180,E1 -2773.947,E2 -2773.947} C_VEL
LIN {X 0,Y 559.157,Z 285.827,A -85,B 0,C 180,E1 -2776.183,E2 -2776.183} C_VEL
LIN {X 0,Y 559.205,Z 285.824,A -85,B 0,C 180,E1 -2778.605,E2 -2778.605} C_VEL
LIN {X 0,Y 559.189,Z 285.826,A -85,B 0,C 180,E1 -2782.053,E2 -2782.053} C_VEL
LIN {X 0,Y 559.258,Z 286.014,A -85,B 0,C 180,E1 -2784.139,E2 -2784.139} C_VEL
LIN {X 0,Y 559.514,Z 291.516,A -85,B 0,C 180,E1 -2785.136,E2 -2785.136} C_VEL
LIN {X 0,Y 559.354,Z 305.748,A -85,B 0,C 180,E1 -2787.659,E2 -2787.659} C_VEL
LIN {X 0,Y 559.261,Z 318.141,A -85,B 0,C 180,E1 -2789.864,E2 -2789.864} C_VEL
LIN {X 0,Y 560.317,Z 325.774,A -85,B 0,C 180,E1 -2789.999,E2 -2789.999} C_VEL
LIN {X 0,Y 560.041,Z 425.58,A -85,B 0,C 180,E1 -2791.303,E2 -2791.303} C_VEL
LIN {X 0,Y 559.872,Z 437.778,A -85,B 0,C 180,E1 -2791.595,E2 -2791.595} C_VEL
LIN {X 0,Y 559.756,Z 450.98,A -85,B 0,C 180,E1 -2792.068,E2 -2792.068} C_VEL
LIN {X 0,Y 559.615,Z 462.133,A -85,B 0,C 180,E1 -2792.609,E2 -2792.609} C_VEL
LIN {X 0,Y 559.439,Z 473.685,A -85,B 0,C 180,E1 -2793.33,E2 -2793.33} C_VEL
LIN {X 0,Y 559.306,Z 484.086,A -85,B 0,C 180,E1 -2794.143,E2 -2794.143} C_VEL
LIN {X 0,Y 559.149,Z 493.485,A -85,B 0,C 180,E1 -2795.047,E2 -2795.047} C_VEL
LIN {X 0,Y 559.035,Z 501.259,A -85,B 0,C 180,E1 -2795.953,E2 -2795.953} C_VEL
LIN {X 0,Y 558.936,Z 508.856,A -85,B 0,C 180,E1 -2797.041,E2 -2797.041} C_VEL
LIN {X 0,Y 558.874,Z 515.894,A -85,B 0,C 180,E1 -2798.314,E2 -2798.314} C_VEL
LIN {X 0,Y 558.803,Z 520.582,A -85,B 0,C 180,E1 -2799.409,E2 -2799.409} C_VEL
LIN {X 0,Y 558.816,Z 524.156,A -85,B 0,C 180,E1 -2800.507,E2 -2800.507} C_VEL
LIN {X 0,Y 558.771,Z 526.716,A -85,B 0,C 180,E1 -2801.609,E2 -2801.609} C_VEL
LIN {X 0,Y 558.77,Z 527.898,A -85,B 0,C 180,E1 -2802.346,E2 -2802.346} C_VEL
LIN {X 0,Y 558.742,Z 528.628,A -85,B 0,C 180,E1 -2803.085,E2 -2803.085} C_VEL
LIN {X 0,Y 558.787,Z 528.921,A -85,B 0,C 180,E1 -2804.432,E2 -2804.432} C_VEL
LIN {X 0,Y 558.715,Z 528.371,A -85,B 0,C 180,E1 -2805.316,E2 -2805.316} C_VEL
LIN {X 0,Y 558.742,Z 527.419,A -85,B 0,C 180,E1 -2806.064,E2 -2806.064} C_VEL
LIN {X 0,Y 558.764,Z 525.447,A -85,B 0,C 180,E1 -2807.078,E2 -2807.078} C_VEL
LIN {X 0,Y 558.813,Z 521.841,A -85,B 0,C 180,E1 -2808.325,E2 -2808.325} C_VEL
LIN {X 0,Y 558.882,Z 516.776,A -85,B 0,C 180,E1 -2809.589,E2 -2809.589} C_VEL
LIN {X 0,Y 558.931,Z 510.351,A -85,B 0,C 180,E1 -2810.806,E2 -2810.806} C_VEL
LIN {X 0,Y 559.043,Z 502.49,A -85,B 0,C 180,E1 -2811.973,E2 -2811.973} C_VEL
LIN {X 0,Y 559.148,Z 494.523,A -85,B 0,C 180,E1 -2812.931,E2 -2812.931} C_VEL
LIN {X 0,Y 559.294,Z 485.667,A -85,B 0,C 180,E1 -2813.807,E2 -2813.807} C_VEL
LIN {X 0,Y 559.38,Z 476.05,A -85,B 0,C 180,E1 -2814.593,E2 -2814.593} C_VEL
LIN {X 0,Y 559.61,Z 463.961,A -85,B 0,C 180,E1 -2815.376,E2 -2815.376} C_VEL
LIN {X 0,Y 559.752,Z 452.251,A -85,B 0,C 180,E1 -2815.967,E2 -2815.967} C_VEL
LIN {X 0,Y 559.875,Z 439.685,A -85,B 0,C 180,E1 -2816.437,E2 -2816.437} C_VEL
LIN {X 0,Y 559.989,Z 427.085,A -85,B 0,C 180,E1 -2816.758,E2 -2816.758} C_VEL
LIN {X 0,Y 560.099,Z 402.728,A -85,B 0,C 180,E1 -2817.102,E2 -2817.102} C_VEL
LIN {X 0,Y 560.195,Z 323.95,A -85,B 0,C 180,E1 -2818.117,E2 -2818.117} C_VEL
LIN {X 0,Y 559.239,Z 318.19,A -85,B 0,C 180,E1 -2818.218,E2 -2818.218} C_VEL
LIN {X 0,Y 559.42,Z 302.487,A -85,B 0,C 180,E1 -2821.002,E2 -2821.002} C_VEL
LIN {X 0,Y 559.498,Z 289.1,A -85,B 0,C 180,E1 -2823.335,E2 -2823.335} C_VEL
LIN {X 0,Y 559.161,Z 285.834,A -85,B 0,C 180,E1 -2823.948,E2 -2823.948} C_VEL
LIN {X 0,Y 559.133,Z 285.838,A -85,B 0,C 180,E1 -2827.108,E2 -2827.108} C_VEL
LIN {X 0,Y 559.151,Z 285.829,A -85,B 0,C 180,E1 -2829.941,E2 -2829.941} C_VEL
LIN {X 0,Y 559.143,Z 285.836,A -85,B 0,C 180,E1 -2832.744,E2 -2832.744} C_VEL
LIN {X 0,Y 559.116,Z 285.835,A -85,B 0,C 180,E1 -2835.763,E2 -2835.763} C_VEL
LIN {X 0,Y 559.117,Z 285.833,A -85,B 0,C 180,E1 -2838.226,E2 -2838.226} C_VEL
LIN {X 0,Y 559.161,Z 285.837,A -85,B 0,C 180,E1 -2841.192,E2 -2841.192} C_VEL
LIN {X 0,Y 559.129,Z 285.835,A -85,B 0,C 180,E1 -2843.789,E2 -2843.789} C_VEL
LIN {X 0,Y 559.136,Z 285.827,A -85,B 0,C 180,E1 -2846.423,E2 -2846.423} C_VEL
LIN {X 0,Y 559.138,Z 285.833,A -85,B 0,C 180,E1 -2848.98,E2 -2848.98} C_VEL
LIN {X 0,Y 559.123,Z 285.842,A -85,B 0,C 180,E1 -2851.625,E2 -2851.625} C_VEL
LIN {X 0,Y 559.128,Z 285.831,A -85,B 0,C 180,E1 -2854.822,E2 -2854.822} C_VEL
LIN {X 0,Y 559.127,Z 285.84,A -85,B 0,C 180,E1 -2857.847,E2 -2857.847} C_VEL
LIN {X 0,Y 559.182,Z 285.826,A -85,B 0,C 180,E1 -2860.494,E2 -2860.494} C_VEL
LIN {X 0,Y 559.11,Z 285.833,A -85,B 0,C 180,E1 -2863.196,E2 -2863.196} C_VEL
LIN {X 0,Y 559.133,Z 285.837,A -85,B 0,C 180,E1 -2866.183,E2 -2866.183} C_VEL
LIN {X 0,Y 559.153,Z 285.828,A -85,B 0,C 180,E1 -2869.133,E2 -2869.133} C_VEL
LIN {X 0,Y 559.127,Z 285.838,A -85,B 0,C 180,E1 -2872.053,E2 -2872.053} C_VEL
LIN {X 0,Y 559.209,Z 285.822,A -85,B 0,C 180,E1 -2874.953,E2 -2874.953} C_VEL
LIN {X 0,Y 559.219,Z 285.821,A -85,B 0,C 180,E1 -2877.839,E2 -2877.839} C_VEL
LIN {X 0,Y 559.257,Z 285.82,A -85,B 0,C 180,E1 -2880.72,E2 -2880.72} C_VEL
LIN {X 0,Y 559.212,Z 285.825,A -85,B 0,C 180,E1 -2882.882,E2 -2882.882} C_VEL
LIN {X 0,Y 559.188,Z 285.824,A -85,B 0,C 180,E1 -2885.771,E2 -2885.771} C_VEL
LIN {X 0,Y 559.125,Z 285.83,A -85,B 0,C 180,E1 -2887.948,E2 -2887.948} C_VEL
LIN {X 0,Y 559.171,Z 285.834,A -85,B 0,C 180,E1 -2890.867,E2 -2890.867} C_VEL
LIN {X 0,Y 559.135,Z 285.828,A -85,B 0,C 180,E1 -2893.817,E2 -2893.817} C_VEL
LIN {X 0,Y 559.144,Z 285.837,A -85,B 0,C 180,E1 -2896.804,E2 -2896.804} C_VEL
LIN {X 0,Y 559.152,Z 285.828,A -85,B 0,C 180,E1 -2899.838,E2 -2899.838} C_VEL
LIN {X 0,Y 559.122,Z 285.831,A -85,B 0,C 180,E1 -2902.154,E2 -2902.154} C_VEL
LIN {X 0,Y 559.13,Z 285.841,A -85,B 0,C 180,E1 -2905.178,E2 -2905.178} C_VEL
LIN {X 0,Y 559.12,Z 285.835,A -85,B 0,C 180,E1 -2907.716,E2 -2907.716} C_VEL
LIN {X 0,Y 559.128,Z 285.832,A -85,B 0,C 180,E1 -2910.185,E2 -2910.185} C_VEL
LIN {X 0,Y 559.148,Z 285.829,A -85,B 0,C 180,E1 -2912.716,E2 -2912.716} C_VEL
LIN {X 0,Y 559.115,Z 285.84,A -85,B 0,C 180,E1 -2915.325,E2 -2915.325} C_VEL
LIN {X 0,Y 559.122,Z 285.835,A -85,B 0,C 180,E1 -2918.019,E2 -2918.019} C_VEL
LIN {X 0,Y 559.149,Z 285.829,A -85,B 0,C 180,E1 -2920.813,E2 -2920.813} C_VEL
LIN {X 0,Y 559.13,Z 285.837,A -85,B 0,C 180,E1 -2923.735,E2 -2923.735} C_VEL
LIN {X 0,Y 559.136,Z 285.831,A -85,B 0,C 180,E1 -2926.805,E2 -2926.805} C_VEL
LIN {X 0,Y 559.151,Z 285.83,A -85,B 0,C 180,E1 -2929.188,E2 -2929.188} C_VEL
LIN {X 0,Y 559.125,Z 285.842,A -85,B 0,C 180,E1 -2931.983,E2 -2931.983} C_VEL
LIN {X 0,Y 559.125,Z 285.832,A -85,B 0,C 180,E1 -2934.789,E2 -2934.789} C_VEL
LIN {X 0,Y 559.153,Z 285.829,A -85,B 0,C 180,E1 -2937.365,E2 -2937.365} C_VEL
LIN {X 0,Y 559.137,Z 285.84,A -85,B 0,C 180,E1 -2940.145,E2 -2940.145} C_VEL
LIN {X 0,Y 559.164,Z 285.829,A -85,B 0,C 180,E1 -2943.175,E2 -2943.175} C_VEL
LIN {X 0,Y 559.124,Z 285.839,A -85,B 0,C 180,E1 -2945.494,E2 -2945.494} C_VEL
LIN {X 0,Y 559.141,Z 285.902,A -85,B 0,C 180,E1 -2946.688,E2 -2946.688} C_VEL
LIN {X 0,Y 560.026,Z 290.997,A -85,B 0,C 180,E1 -2947.496,E2 -2947.496} C_VEL
LIN {X 0,Y 559.832,Z 308.916,A -85,B 0,C 180,E1 -2950.188,E2 -2950.188} C_VEL
LIN {X 0,Y 559.602,Z 327.408,A -85,B 0,C 180,E1 -2952.926,E2 -2952.926} C_VEL
LIN {X 0,Y 559.392,Z 347.202,A -85,B 0,C 180,E1 -2955.819,E2 -2955.819} C_VEL
LIN {X 0,Y 560.289,Z 354.357,A -85,B 0,C 180,E1 -2955.935,E2 -2955.935} C_VEL
LIN {X 0,Y 560.073,Z 454.984,A -85,B 0,C 180,E1 -2957.246,E2 -2957.246} C_VEL
LIN {X 0,Y 559.915,Z 468.242,A -85,B 0,C 180,E1 -2957.565,E2 -2957.565} C_VEL
LIN {X 0,Y 559.765,Z 481.514,A -85,B 0,C 180,E1 -2958.045,E2 -2958.045} C_VEL
LIN {X 0,Y 559.64,Z 493.776,A -85,B 0,C 180,E1 -2958.659,E2 -2958.659} C_VEL
LIN {X 0,Y 559.431,Z 505.496,A -85,B 0,C 180,E1 -2959.414,E2 -2959.414} C_VEL
LIN {X 0,Y 559.288,Z 515.622,A -85,B 0,C 180,E1 -2960.234,E2 -2960.234} C_VEL
LIN {X 0,Y 559.132,Z 524.792,A -85,B 0,C 180,E1 -2961.143,E2 -2961.143} C_VEL
LIN {X 0,Y 559.009,Z 533.694,A -85,B 0,C 180,E1 -2962.233,E2 -2962.233} C_VEL
LIN {X 0,Y 558.936,Z 541.214,A -85,B 0,C 180,E1 -2963.385,E2 -2963.385} C_VEL
LIN {X 0,Y 558.869,Z 547.369,A -85,B 0,C 180,E1 -2964.589,E2 -2964.589} C_VEL
LIN {X 0,Y 558.868,Z 551.679,A -85,B 0,C 180,E1 -2965.673,E2 -2965.673} C_VEL
LIN {X 0,Y 558.836,Z 553.96,A -85,B 0,C 180,E1 -2966.396,E2 -2966.396} C_VEL
LIN {X 0,Y 558.799,Z 555.809,A -85,B 0,C 180,E1 -2967.117,E2 -2967.117} C_VEL
LIN {X 0,Y 558.745,Z 558.185,A -85,B 0,C 180,E1 -2968.559,E2 -2968.559} C_VEL
LIN {X 0,Y 558.74,Z 559,A -85,B 0,C 180,E1 -2970.001,E2 -2970.001} C_VEL
LIN {X 0,Y 558.745,Z 558.184,A -85,B 0,C 180,E1 -2971.442,E2 -2971.442} C_VEL
LIN {X 0,Y 558.8,Z 555.809,A -85,B 0,C 180,E1 -2972.884,E2 -2972.884} C_VEL
LIN {X 0,Y 558.844,Z 552.894,A -85,B 0,C 180,E1 -2973.967,E2 -2973.967} C_VEL
LIN {X 0,Y 558.798,Z 548.946,A -85,B 0,C 180,E1 -2975.051,E2 -2975.051} C_VEL
LIN {X 0,Y 558.925,Z 543.864,A -85,B 0,C 180,E1 -2976.136,E2 -2976.136} C_VEL
LIN {X 0,Y 558.975,Z 537.463,A -85,B 0,C 180,E1 -2977.224,E2 -2977.224} C_VEL
LIN {X 0,Y 559.092,Z 529.473,A -85,B 0,C 180,E1 -2978.312,E2 -2978.312} C_VEL
LIN {X 0,Y 559.198,Z 521.328,A -85,B 0,C 180,E1 -2979.222,E2 -2979.222} C_VEL
LIN {X 0,Y 559.344,Z 511.392,A -85,B 0,C 180,E1 -2980.132,E2 -2980.132} C_VEL
LIN {X 0,Y 559.571,Z 500.39,A -85,B 0,C 180,E1 -2980.937,E2 -2980.937} C_VEL
LIN {X 0,Y 559.673,Z 488.448,A -85,B 0,C 180,E1 -2981.628,E2 -2981.628} C_VEL
LIN {X 0,Y 559.834,Z 475.751,A -85,B 0,C 180,E1 -2982.185,E2 -2982.185} C_VEL
LIN {X 0,Y 559.946,Z 462.322,A -85,B 0,C 180,E1 -2982.597,E2 -2982.597} C_VEL
LIN {X 0,Y 560.069,Z 449.043,A -85,B 0,C 180,E1 -2982.847,E2 -2982.847} C_VEL
LIN {X 0,Y 560.194,Z 352.264,A -85,B 0,C 180,E1 -2984.094,E2 -2984.094} C_VEL
LIN {X 0,Y 559.369,Z 346.788,A -85,B 0,C 180,E1 -2984.206,E2 -2984.206} C_VEL
LIN {X 0,Y 559.606,Z 327.386,A -85,B 0,C 180,E1 -2987.077,E2 -2987.077} C_VEL
LIN {X 0,Y 559.862,Z 307.69,A -85,B 0,C 180,E1 -2990.004,E2 -2990.004} C_VEL
LIN {X 0,Y 560.039,Z 291.104,A -85,B 0,C 180,E1 -2992.505,E2 -2992.505} C_VEL
LIN {X 0,Y 559.12,Z 285.843,A -85,B 0,C 180,E1 -2993.386,E2 -2993.386} C_VEL
LIN {X 0,Y 559.175,Z 285.83,A -85,B 0,C 180,E1 -2996.098,E2 -2996.098} C_VEL
LIN {X 0,Y 559.14,Z 285.831,A -85,B 0,C 180,E1 -2998.531,E2 -2998.531} C_VEL
LIN {X 0,Y 559.145,Z 285.831,A -85,B 0,C 180,E1 -3001.273,E2 -3001.273} C_VEL
LIN {X 0,Y 559.168,Z 285.837,A -85,B 0,C 180,E1 -3003.949,E2 -3003.949} C_VEL
LIN {X 0,Y 559.134,Z 285.83,A -85,B 0,C 180,E1 -3007.109,E2 -3007.109} C_VEL
LIN {X 0,Y 559.163,Z 285.833,A -85,B 0,C 180,E1 -3009.942,E2 -3009.942} C_VEL
LIN {X 0,Y 559.151,Z 285.831,A -85,B 0,C 180,E1 -3012.745,E2 -3012.745} C_VEL
LIN {X 0,Y 559.151,Z 285.829,A -85,B 0,C 180,E1 -3015.762,E2 -3015.762} C_VEL
LIN {X 0,Y 559.164,Z 285.832,A -85,B 0,C 180,E1 -3018.23,E2 -3018.23} C_VEL
LIN {X 0,Y 559.175,Z 285.827,A -85,B 0,C 180,E1 -3021.192,E2 -3021.192} C_VEL
LIN {X 0,Y 559.124,Z 285.831,A -85,B 0,C 180,E1 -3023.788,E2 -3023.788} C_VEL
LIN {X 0,Y 559.163,Z 285.83,A -85,B 0,C 180,E1 -3026.425,E2 -3026.425} C_VEL
LIN {X 0,Y 559.153,Z 285.838,A -85,B 0,C 180,E1 -3028.98,E2 -3028.98} C_VEL
LIN {X 0,Y 559.149,Z 285.83,A -85,B 0,C 180,E1 -3031.623,E2 -3031.623} C_VEL
LIN {X 0,Y 559.164,Z 285.827,A -85,B 0,C 180,E1 -3033.902,E2 -3033.902} C_VEL
LIN {X 0,Y 559.12,Z 285.84,A -85,B 0,C 180,E1 -3037.066,E2 -3037.066} C_VEL
LIN {X 0,Y 559.178,Z 285.834,A -85,B 0,C 180,E1 -3039.395,E2 -3039.395} C_VEL
LIN {X 0,Y 559.141,Z 285.835,A -85,B 0,C 180,E1 -3041.685,E2 -3041.685} C_VEL
LIN {X 0,Y 559.164,Z 285.83,A -85,B 0,C 180,E1 -3043.948,E2 -3043.948} C_VEL
LIN {X 0,Y 559.166,Z 285.828,A -85,B 0,C 180,E1 -3046.184,E2 -3046.184} C_VEL
LIN {X 0,Y 559.196,Z 285.824,A -85,B 0,C 180,E1 -3049.133,E2 -3049.133} C_VEL
LIN {X 0,Y 559.173,Z 285.832,A -85,B 0,C 180,E1 -3052.053,E2 -3052.053} C_VEL
LIN {X 0,Y 559.249,Z 285.816,A -85,B 0,C 180,E1 -3054.953,E2 -3054.953} C_VEL
LIN {X 0,Y 559.257,Z 285.822,A -85,B 0,C 180,E1 -3057.839,E2 -3057.839} C_VEL
LIN {X 0,Y 559.263,Z 285.816,A -85,B 0,C 180,E1 -3060.72,E2 -3060.72} C_VEL
LIN {X 0,Y 559.229,Z 285.82,A -85,B 0,C 180,E1 -3062.881,E2 -3062.881} C_VEL
LIN {X 0,Y 559.217,Z 285.822,A -85,B 0,C 180,E1 -3065.77,E2 -3065.77} C_VEL
LIN {X 0,Y 559.185,Z 285.83,A -85,B 0,C 180,E1 -3068.674,E2 -3068.674} C_VEL
LIN {X 0,Y 559.208,Z 285.821,A -85,B 0,C 180,E1 -3071.6,E2 -3071.6} C_VEL
LIN {X 0,Y 559.204,Z 285.831,A -85,B 0,C 180,E1 -3074.595,E2 -3074.595} C_VEL
LIN {X 0,Y 559.141,Z 285.83,A -85,B 0,C 180,E1 -3077.557,E2 -3077.557} C_VEL
LIN {X 0,Y 559.167,Z 285.826,A -85,B 0,C 180,E1 -3079.837,E2 -3079.837} C_VEL
LIN {X 0,Y 559.141,Z 285.83,A -85,B 0,C 180,E1 -3082.153,E2 -3082.153} C_VEL
LIN {X 0,Y 559.176,Z 285.832,A -85,B 0,C 180,E1 -3085.298,E2 -3085.298} C_VEL
LIN {X 0,Y 559.131,Z 285.833,A -85,B 0,C 180,E1 -3087.715,E2 -3087.715} C_VEL
LIN {X 0,Y 559.135,Z 285.831,A -85,B 0,C 180,E1 -3090.607,E2 -3090.607} C_VEL
LIN {X 0,Y 558.473,Z 285.922,A -85,B 0,C 180,E1 -3091.208,E2 -3091.208} C_VEL
LIN {X 0,Y 555.611,Z 286.275,A -85,B 0,C 180,E1 -3092.184,E2 -3092.184} C_VEL
LIN {X 0,Y 553.195,Z 286.574,A -85,B 0,C 180,E1 -3092.97,E2 -3092.97} C_VEL
LIN {X 0,Y 552.169,Z 286.705,A -85,B 0,C 180,E1 -3093.576,E2 -3093.576} C_VEL
LIN {X 0,Y 552.091,Z 286.709,A -85,B 0,C 180,E1 -3093.782,E2 -3093.782} C_VEL
LIN {X 0,Y 552.1,Z 286.707,A -85,B 0,C 180,E1 -3096.747,E2 -3096.747} C_VEL
LIN {X 0,Y 552.132,Z 286.711,A -85,B 0,C 180,E1 -3099.527,E2 -3099.527} C_VEL
LIN {X 0,Y 552.11,Z 286.706,A -85,B 0,C 180,E1 -3102.427,E2 -3102.427} C_VEL
LIN {X 0,Y 552.096,Z 286.712,A -85,B 0,C 180,E1 -3105.562,E2 -3105.562} C_VEL
LIN {X 0,Y 552.122,Z 286.705,A -85,B 0,C 180,E1 -3108.678,E2 -3108.678} C_VEL
LIN {X 0,Y 552.114,Z 286.706,A -85,B 0,C 180,E1 -3111.41,E2 -3111.41} C_VEL
LIN {X 0,Y 552.076,Z 286.72,A -85,B 0,C 180,E1 -3114.155,E2 -3114.155} C_VEL
LIN {X 0,Y 552.115,Z 286.707,A -85,B 0,C 180,E1 -3116.814,E2 -3116.814} C_VEL
LIN {X 0,Y 552.102,Z 286.706,A -85,B 0,C 180,E1 -3119.39,E2 -3119.39} C_VEL
LIN {X 0,Y 552.089,Z 286.71,A -85,B 0,C 180,E1 -3121.9,E2 -3121.9} C_VEL
LIN {X 0,Y 552.087,Z 286.717,A -85,B 0,C 180,E1 -3124.665,E2 -3124.665} C_VEL
LIN {X 0,Y 552.087,Z 286.708,A -85,B 0,C 180,E1 -3127.548,E2 -3127.548} C_VEL
LIN {X 0,Y 552.145,Z 286.704,A -85,B 0,C 180,E1 -3130.375,E2 -3130.375} C_VEL
LIN {X 0,Y 552.123,Z 286.713,A -85,B 0,C 180,E1 -3132.976,E2 -3132.976} C_VEL
LIN {X 0,Y 552.121,Z 286.704,A -85,B 0,C 180,E1 -3136.004,E2 -3136.004} C_VEL
LIN {X 0,Y 552.154,Z 286.708,A -85,B 0,C 180,E1 -3138.993,E2 -3138.993} C_VEL
LIN {X 0,Y 552.144,Z 286.705,A -85,B 0,C 180,E1 -3141.951,E2 -3141.951} C_VEL
LIN {X 0,Y 552.207,Z 286.745,A -85,B 0,C 180,E1 -3144.018,E2 -3144.018} C_VEL
LIN {X 0,Y 552.473,Z 291.513,A -85,B 0,C 180,E1 -3144.891,E2 -3144.891} C_VEL
LIN {X 0,Y 552.383,Z 304.764,A -85,B 0,C 180,E1 -3147.265,E2 -3147.265} C_VEL
LIN {X 0,Y 552.235,Z 318.174,A -85,B 0,C 180,E1 -3149.68,E2 -3149.68} C_VEL
LIN {X 0,Y 553.415,Z 325.569,A -85,B 0,C 180,E1 -3149.817,E2 -3149.817} C_VEL
LIN {X 0,Y 553.142,Z 425.376,A -85,B 0,C 180,E1 -3151.137,E2 -3151.137} C_VEL
LIN {X 0,Y 552.959,Z 437.646,A -85,B 0,C 180,E1 -3151.433,E2 -3151.433} C_VEL
LIN {X 0,Y 552.796,Z 450.905,A -85,B 0,C 180,E1 -3151.912,E2 -3151.912} C_VEL
LIN {X 0,Y 552.634,Z 462.082,A -85,B 0,C 180,E1 -3152.459,E2 -3152.459} C_VEL
LIN {X 0,Y 552.441,Z 473.642,A -85,B 0,C 180,E1 -3153.19,E2 -3153.19} C_VEL
LIN {X 0,Y 552.278,Z 484.054,A -85,B 0,C 180,E1 -3154.013,E2 -3154.013} C_VEL
LIN {X 0,Y 552.121,Z 493.471,A -85,B 0,C 180,E1 -3154.928,E2 -3154.928} C_VEL
LIN {X 0,Y 551.976,Z 502.473,A -85,B 0,C 180,E1 -3156.013,E2 -3156.013} C_VEL
LIN {X 0,Y 551.866,Z 509.953,A -85,B 0,C 180,E1 -3157.132,E2 -3157.132} C_VEL
LIN {X 0,Y 551.775,Z 516.744,A -85,B 0,C 180,E1 -3158.422,E2 -3158.422} C_VEL
LIN {X 0,Y 551.728,Z 521.234,A -85,B 0,C 180,E1 -3159.531,E2 -3159.531} C_VEL
LIN {X 0,Y 551.716,Z 523.608,A -85,B 0,C 180,E1 -3160.272,E2 -3160.272} C_VEL
LIN {X 0,Y 551.719,Z 526.027,A -85,B 0,C 180,E1 -3161.23,E2 -3161.23} C_VEL
LIN {X 0,Y 551.656,Z 528.099,A -85,B 0,C 180,E1 -3162.507,E2 -3162.507} C_VEL
LIN {X 0,Y 551.655,Z 528.748,A -85,B 0,C 180,E1 -3163.256,E2 -3163.256} C_VEL
LIN {X 0,Y 551.692,Z 528.908,A -85,B 0,C 180,E1 -3164.497,E2 -3164.497} C_VEL
LIN {X 0,Y 551.614,Z 528.169,A -85,B 0,C 180,E1 -3165.518,E2 -3165.518} C_VEL
LIN {X 0,Y 551.649,Z 527.132,A -85,B 0,C 180,E1 -3166.276,E2 -3166.276} C_VEL
LIN {X 0,Y 551.682,Z 525.32,A -85,B 0,C 180,E1 -3167.169,E2 -3167.169} C_VEL
LIN {X 0,Y 551.716,Z 521.2,A -85,B 0,C 180,E1 -3168.569,E2 -3168.569} C_VEL
LIN {X 0,Y 551.81,Z 516.402,A -85,B 0,C 180,E1 -3169.744,E2 -3169.744} C_VEL
LIN {X 0,Y 551.859,Z 510.37,A -85,B 0,C 180,E1 -3170.89,E2 -3170.89} C_VEL
LIN {X 0,Y 551.972,Z 502.592,A -85,B 0,C 180,E1 -3172.061,E2 -3172.061} C_VEL
LIN {X 0,Y 552.088,Z 494.547,A -85,B 0,C 180,E1 -3173.043,E2 -3173.043} C_VEL
LIN {X 0,Y 552.252,Z 484.603,A -85,B 0,C 180,E1 -3174.03,E2 -3174.03} C_VEL
LIN {X 0,Y 552.446,Z 473.502,A -85,B 0,C 180,E1 -3174.91,E2 -3174.91} C_VEL
LIN {X 0,Y 552.665,Z 462.314,A -85,B 0,C 180,E1 -3175.617,E2 -3175.617} C_VEL
LIN {X 0,Y 552.813,Z 449.97,A -85,B 0,C 180,E1 -3176.217,E2 -3176.217} C_VEL
LIN {X 0,Y 552.979,Z 436.519,A -85,B 0,C 180,E1 -3176.691,E2 -3176.691} C_VEL
LIN {X 0,Y 553.145,Z 423.404,A -85,B 0,C 180,E1 -3176.988,E2 -3176.988} C_VEL
LIN {X 0,Y 553.268,Z 324.457,A -85,B 0,C 180,E1 -3178.291,E2 -3178.291} C_VEL
LIN {X 0,Y 552.228,Z 318.134,A -85,B 0,C 180,E1 -3178.418,E2 -3178.418} C_VEL
LIN {X 0,Y 552.416,Z 301.129,A -85,B 0,C 180,E1 -3181.44,E2 -3181.44} C_VEL
LIN {X 0,Y 552.382,Z 288.672,A -85,B 0,C 180,E1 -3183.603,E2 -3183.603} C_VEL
LIN {X 0,Y 552.121,Z 286.711,A -85,B 0,C 180,E1 -3183.978,E2 -3183.978} C_VEL
LIN {X 0,Y 552.099,Z 286.717,A -85,B 0,C 180,E1 -3186.746,E2 -3186.746} C_VEL
LIN {X 0,Y 552.12,Z 286.707,A -85,B 0,C 180,E1 -3189.527,E2 -3189.527} C_VEL
LIN {X 0,Y 552.102,Z 286.709,A -85,B 0,C 180,E1 -3192.427,E2 -3192.427} C_VEL
LIN {X 0,Y 552.067,Z 286.715,A -85,B 0,C 180,E1 -3195.56,E2 -3195.56} C_VEL
LIN {X 0,Y 552.066,Z 286.712,A -85,B 0,C 180,E1 -3198.549,E2 -3198.549} C_VEL
LIN {X 0,Y 552.105,Z 286.714,A -85,B 0,C 180,E1 -3201.41,E2 -3201.41} C_VEL
LIN {X 0,Y 552.076,Z 286.711,A -85,B 0,C 180,E1 -3204.156,E2 -3204.156} C_VEL
LIN {X 0,Y 552.096,Z 286.705,A -85,B 0,C 180,E1 -3206.813,E2 -3206.813} C_VEL
LIN {X 0,Y 552.082,Z 286.718,A -85,B 0,C 180,E1 -3209.39,E2 -3209.39} C_VEL
LIN {X 0,Y 552.066,Z 286.717,A -85,B 0,C 180,E1 -3211.899,E2 -3211.899} C_VEL
LIN {X 0,Y 552.069,Z 286.71,A -85,B 0,C 180,E1 -3214.666,E2 -3214.666} C_VEL
LIN {X 0,Y 552.078,Z 286.716,A -85,B 0,C 180,E1 -3217.549,E2 -3217.549} C_VEL
LIN {X 0,Y 552.134,Z 286.705,A -85,B 0,C 180,E1 -3220.375,E2 -3220.375} C_VEL
LIN {X 0,Y 552.072,Z 286.709,A -85,B 0,C 180,E1 -3222.975,E2 -3222.975} C_VEL
LIN {X 0,Y 552.096,Z 286.716,A -85,B 0,C 180,E1 -3226.004,E2 -3226.004} C_VEL
LIN {X 0,Y 552.115,Z 286.705,A -85,B 0,C 180,E1 -3228.993,E2 -3228.993} C_VEL
LIN {X 0,Y 552.096,Z 286.711,A -85,B 0,C 180,E1 -3231.951,E2 -3231.951} C_VEL
LIN {X 0,Y 552.186,Z 286.697,A -85,B 0,C 180,E1 -3234.889,E2 -3234.889} C_VEL
LIN {X 0,Y 552.192,Z 286.695,A -85,B 0,C 180,E1 -3237.812,E2 -3237.812} C_VEL
LIN {X 0,Y 552.227,Z 286.695,A -85,B 0,C 180,E1 -3240.729,E2 -3240.729} C_VEL
LIN {X 0,Y 552.177,Z 286.7,A -85,B 0,C 180,E1 -3242.918,E2 -3242.918} C_VEL
LIN {X 0,Y 552.161,Z 286.7,A -85,B 0,C 180,E1 -3245.844,E2 -3245.844} C_VEL
LIN {X 0,Y 552.116,Z 286.714,A -85,B 0,C 180,E1 -3248.787,E2 -3248.787} C_VEL
LIN {X 0,Y 552.142,Z 286.7,A -85,B 0,C 180,E1 -3251.751,E2 -3251.751} C_VEL
LIN {X 0,Y 552.11,Z 286.712,A -85,B 0,C 180,E1 -3254.749,E2 -3254.749} C_VEL
LIN {X 0,Y 552.08,Z 286.707,A -85,B 0,C 180,E1 -3257.79,E2 -3257.79} C_VEL
LIN {X 0,Y 552.114,Z 286.704,A -85,B 0,C 180,E1 -3260.102,E2 -3260.102} C_VEL
LIN {X 0,Y 552.074,Z 286.71,A -85,B 0,C 180,E1 -3262.452,E2 -3262.452} C_VEL
LIN {X 0,Y 552.075,Z 286.718,A -85,B 0,C 180,E1 -3265.335,E2 -3265.335} C_VEL
LIN {X 0,Y 552.069,Z 286.71,A -85,B 0,C 180,E1 -3268.101,E2 -3268.101} C_VEL
LIN {X 0,Y 552.084,Z 286.709,A -85,B 0,C 180,E1 -3270.611,E2 -3270.611} C_VEL
LIN {X 0,Y 552.108,Z 286.711,A -85,B 0,C 180,E1 -3273.187,E2 -3273.187} C_VEL
LIN {X 0,Y 552.067,Z 286.716,A -85,B 0,C 180,E1 -3275.845,E2 -3275.845} C_VEL
LIN {X 0,Y 552.108,Z 286.705,A -85,B 0,C 180,E1 -3278.59,E2 -3278.59} C_VEL
LIN {X 0,Y 552.107,Z 286.713,A -85,B 0,C 180,E1 -3281.448,E2 -3281.448} C_VEL
LIN {X 0,Y 552.083,Z 286.71,A -85,B 0,C 180,E1 -3284.532,E2 -3284.532} C_VEL
LIN {X 0,Y 552.105,Z 286.713,A -85,B 0,C 180,E1 -3287.588,E2 -3287.588} C_VEL
LIN {X 0,Y 552.124,Z 286.708,A -85,B 0,C 180,E1 -3290.474,E2 -3290.474} C_VEL
LIN {X 0,Y 552.095,Z 286.709,A -85,B 0,C 180,E1 -3293.319,E2 -3293.319} C_VEL
LIN {X 0,Y 552.122,Z 286.711,A -85,B 0,C 180,E1 -3295.94,E2 -3295.94} C_VEL
LIN {X 0,Y 552.118,Z 286.711,A -85,B 0,C 180,E1 -3298.542,E2 -3298.542} C_VEL
LIN {X 0,Y 552.101,Z 286.708,A -85,B 0,C 180,E1 -3301.443,E2 -3301.443} C_VEL
LIN {X 0,Y 552.112,Z 286.708,A -85,B 0,C 180,E1 -3303.544,E2 -3303.544} C_VEL
LIN {X 0,Y 552.124,Z 286.805,A -85,B 0,C 180,E1 -3306.551,E2 -3306.551} C_VEL
LIN {X 0,Y 553.078,Z 293.327,A -85,B 0,C 180,E1 -3307.592,E2 -3307.592} C_VEL
LIN {X 0,Y 552.813,Z 312.06,A -85,B 0,C 180,E1 -3310.436,E2 -3310.436} C_VEL
LIN {X 0,Y 552.572,Z 329.117,A -85,B 0,C 180,E1 -3312.991,E2 -3312.991} C_VEL
LIN {X 0,Y 552.355,Z 346.905,A -85,B 0,C 180,E1 -3315.628,E2 -3315.628} C_VEL
LIN {X 0,Y 553.402,Z 354.946,A -85,B 0,C 180,E1 -3315.764,E2 -3315.764} C_VEL
LIN {X 0,Y 553.161,Z 454.984,A -85,B 0,C 180,E1 -3317.084,E2 -3317.084} C_VEL
LIN {X 0,Y 552.994,Z 468.242,A -85,B 0,C 180,E1 -3317.407,E2 -3317.407} C_VEL
LIN {X 0,Y 552.835,Z 481.176,A -85,B 0,C 180,E1 -3317.879,E2 -3317.879} C_VEL
LIN {X 0,Y 552.683,Z 493.639,A -85,B 0,C 180,E1 -3318.506,E2 -3318.506} C_VEL
LIN {X 0,Y 552.453,Z 505.496,A -85,B 0,C 180,E1 -3319.278,E2 -3319.278} C_VEL
LIN {X 0,Y 552.274,Z 515.638,A -85,B 0,C 180,E1 -3320.109,E2 -3320.109} C_VEL
LIN {X 0,Y 552.105,Z 524.792,A -85,B 0,C 180,E1 -3321.03,E2 -3321.03} C_VEL
LIN {X 0,Y 551.959,Z 533.693,A -85,B 0,C 180,E1 -3322.134,E2 -3322.134} C_VEL
LIN {X 0,Y 551.861,Z 539.744,A -85,B 0,C 180,E1 -3323.052,E2 -3323.052} C_VEL
LIN {X 0,Y 551.868,Z 545.683,A -85,B 0,C 180,E1 -3324.153,E2 -3324.153} C_VEL
LIN {X 0,Y 551.725,Z 550.376,A -85,B 0,C 180,E1 -3325.251,E2 -3325.251} C_VEL
LIN {X 0,Y 551.751,Z 553.96,A -85,B 0,C 180,E1 -3326.349,E2 -3326.349} C_VEL
LIN {X 0,Y 551.724,Z 555.809,A -85,B 0,C 180,E1 -3327.08,E2 -3327.08} C_VEL
LIN {X 0,Y 551.645,Z 558.184,A -85,B 0,C 180,E1 -3328.541,E2 -3328.541} C_VEL
LIN {X 0,Y 551.64,Z 559,A -85,B 0,C 180,E1 -3330.001,E2 -3330.001} C_VEL
LIN {X 0,Y 551.645,Z 558.184,A -85,B 0,C 180,E1 -3331.461,E2 -3331.461} C_VEL
LIN {X 0,Y 551.724,Z 555.809,A -85,B 0,C 180,E1 -3332.921,E2 -3332.921} C_VEL
LIN {X 0,Y 551.764,Z 552.893,A -85,B 0,C 180,E1 -3334.018,E2 -3334.018} C_VEL
LIN {X 0,Y 551.724,Z 548.946,A -85,B 0,C 180,E1 -3335.116,E2 -3335.116} C_VEL
LIN {X 0,Y 551.826,Z 543.182,A -85,B 0,C 180,E1 -3336.343,E2 -3336.343} C_VEL
LIN {X 0,Y 551.927,Z 536.232,A -85,B 0,C 180,E1 -3337.5,E2 -3337.5} C_VEL
LIN {X 0,Y 552.064,Z 527.987,A -85,B 0,C 180,E1 -3338.603,E2 -3338.603} C_VEL
LIN {X 0,Y 552.22,Z 519.533,A -85,B 0,C 180,E1 -3339.524,E2 -3339.524} C_VEL
LIN {X 0,Y 552.399,Z 509.085,A -85,B 0,C 180,E1 -3340.446,E2 -3340.446} C_VEL
LIN {X 0,Y 552.611,Z 498.277,A -85,B 0,C 180,E1 -3341.214,E2 -3341.214} C_VEL
LIN {X 0,Y 552.754,Z 487.393,A -85,B 0,C 180,E1 -3341.831,E2 -3341.831} C_VEL
LIN {X 0,Y 552.902,Z 475.748,A -85,B 0,C 180,E1 -3342.34,E2 -3342.34} C_VEL
LIN {X 0,Y 553.039,Z 462.321,A -85,B 0,C 180,E1 -3342.757,E2 -3342.757} C_VEL
LIN {X 0,Y 553.172,Z 449.043,A -85,B 0,C 180,E1 -3343.01,E2 -3343.01} C_VEL
LIN {X 0,Y 553.398,Z 353.634,A -85,B 0,C 180,E1 -3344.253,E2 -3344.253} C_VEL
LIN {X 0,Y 552.376,Z 346.766,A -85,B 0,C 180,E1 -3344.392,E2 -3344.392} C_VEL
LIN {X 0,Y 552.642,Z 325.954,A -85,B 0,C 180,E1 -3347.487,E2 -3347.487} C_VEL
LIN {X 0,Y 553.004,Z 304.953,A -85,B 0,C 180,E1 -3350.651,E2 -3350.651} C_VEL
LIN {X 0,Y 553.069,Z 292.205,A -85,B 0,C 180,E1 -3352.607,E2 -3352.607} C_VEL
LIN {X 0,Y 552.089,Z 286.718,A -85,B 0,C 180,E1 -3353.535,E2 -3353.535} C_VEL
LIN {X 0,Y 552.117,Z 286.706,A -85,B 0,C 180,E1 -3356.457,E2 -3356.457} C_VEL
LIN {X 0,Y 552.093,Z 286.708,A -85,B 0,C 180,E1 -3358.93,E2 -3358.93} C_VEL
LIN {X 0,Y 552.116,Z 286.709,A -85,B 0,C 180,E1 -3361.476,E2 -3361.476} C_VEL
LIN {X 0,Y 552.134,Z 286.709,A -85,B 0,C 180,E1 -3364.17,E2 -3364.17} C_VEL
LIN {X 0,Y 552.102,Z 286.707,A -85,B 0,C 180,E1 -3366.748,E2 -3366.748} C_VEL
LIN {X 0,Y 552.131,Z 286.704,A -85,B 0,C 180,E1 -3369.528,E2 -3369.528} C_VEL
LIN {X 0,Y 552.112,Z 286.713,A -85,B 0,C 180,E1 -3372.428,E2 -3372.428} C_VEL
LIN {X 0,Y 552.095,Z 286.707,A -85,B 0,C 180,E1 -3375.562,E2 -3375.562} C_VEL
LIN {X 0,Y 552.124,Z 286.711,A -85,B 0,C 180,E1 -3378.679,E2 -3378.679} C_VEL
LIN {X 0,Y 552.118,Z 286.705,A -85,B 0,C 180,E1 -3381.411,E2 -3381.411} C_VEL
LIN {X 0,Y 552.078,Z 286.711,A -85,B 0,C 180,E1 -3384.155,E2 -3384.155} C_VEL
LIN {X 0,Y 552.116,Z 286.715,A -85,B 0,C 180,E1 -3386.814,E2 -3386.814} C_VEL
LIN {X 0,Y 552.101,Z 286.71,A -85,B 0,C 180,E1 -3389.39,E2 -3389.39} C_VEL
LIN {X 0,Y 552.092,Z 286.707,A -85,B 0,C 180,E1 -3391.9,E2 -3391.9} C_VEL
LIN {X 0,Y 552.086,Z 286.711,A -85,B 0,C 180,E1 -3394.666,E2 -3394.666} C_VEL
LIN {X 0,Y 552.091,Z 286.713,A -85,B 0,C 180,E1 -3397.549,E2 -3397.549} C_VEL
LIN {X 0,Y 552.148,Z 286.7,A -85,B 0,C 180,E1 -3400.375,E2 -3400.375} C_VEL
LIN {X 0,Y 552.137,Z 286.705,A -85,B 0,C 180,E1 -3402.976,E2 -3402.976} C_VEL
LIN {X 0,Y 552.132,Z 286.706,A -85,B 0,C 180,E1 -3406.004,E2 -3406.004} C_VEL
LIN {X 0,Y 552.164,Z 286.699,A -85,B 0,C 180,E1 -3408.993,E2 -3408.993} C_VEL
LIN {X 0,Y 552.134,Z 286.71,A -85,B 0,C 180,E1 -3411.951,E2 -3411.951} C_VEL
LIN {X 0,Y 552.224,Z 286.691,A -85,B 0,C 180,E1 -3414.889,E2 -3414.889} C_VEL
LIN {X 0,Y 552.228,Z 286.697,A -85,B 0,C 180,E1 -3417.812,E2 -3417.812} C_VEL
LIN {X 0,Y 552.235,Z 286.691,A -85,B 0,C 180,E1 -3420.729,E2 -3420.729} C_VEL
LIN {X 0,Y 552.196,Z 286.695,A -85,B 0,C 180,E1 -3422.918,E2 -3422.918} C_VEL
LIN {X 0,Y 552.187,Z 286.698,A -85,B 0,C 180,E1 -3425.844,E2 -3425.844} C_VEL
LIN {X 0,Y 552.152,Z 286.705,A -85,B 0,C 180,E1 -3428.786,E2 -3428.786} C_VEL
LIN {X 0,Y 552.165,Z 286.699,A -85,B 0,C 180,E1 -3431.75,E2 -3431.75} C_VEL
LIN {X 0,Y 552.139,Z 286.711,A -85,B 0,C 180,E1 -3434.748,E2 -3434.748} C_VEL
LIN {X 0,Y 552.099,Z 286.706,A -85,B 0,C 180,E1 -3437.789,E2 -3437.789} C_VEL
LIN {X 0,Y 552.128,Z 286.703,A -85,B 0,C 180,E1 -3440.101,E2 -3440.101} C_VEL
LIN {X 0,Y 552.092,Z 286.71,A -85,B 0,C 180,E1 -3442.451,E2 -3442.451} C_VEL
LIN {X 0,Y 552.139,Z 286.707,A -85,B 0,C 180,E1 -3445.346,E2 -3445.346} C_VEL
LIN {X 0,Y 552.08,Z 286.709,A -85,B 0,C 180,E1 -3448.1,E2 -3448.1} C_VEL
LIN {X 0,Y 552.099,Z 286.708,A -85,B 0,C 180,E1 -3450.609,E2 -3450.609} C_VEL
LIN {X 0,Y 552.108,Z 286.713,A -85,B 0,C 180,E1 -3453.186,E2 -3453.186} C_VEL
LIN {X 0,Y 552.091,Z 286.709,A -85,B 0,C 180,E1 -3453.782,E2 -3453.782} C_VEL
LIN {X 0,Y 551.451,Z 286.79,A -85,B 0,C 180,E1 -3454.39,E2 -3454.39} C_VEL
LIN {X 0,Y 548.635,Z 287.147,A -85,B 0,C 180,E1 -3455.379,E2 -3455.379} C_VEL
LIN {X 0,Y 546.224,Z 287.442,A -85,B 0,C 180,E1 -3456.174,E2 -3456.174} C_VEL
LIN {X 0,Y 545.16,Z 287.572,A -85,B 0,C 180,E1 -3456.788,E2 -3456.788} C_VEL
LIN {X 0,Y 545.059,Z 287.586,A -85,B 0,C 180,E1 -3456.996,E2 -3456.996} C_VEL
LIN {X 0,Y 545.068,Z 287.585,A -85,B 0,C 180,E1 -3460.142,E2 -3460.142} C_VEL
LIN {X 0,Y 545.046,Z 287.586,A -85,B 0,C 180,E1 -3463.11,E2 -3463.11} C_VEL
LIN {X 0,Y 545.051,Z 287.589,A -85,B 0,C 180,E1 -3466.226,E2 -3466.226} C_VEL
LIN {X 0,Y 545.082,Z 287.581,A -85,B 0,C 180,E1 -3468.885,E2 -3468.885} C_VEL
LIN {X 0,Y 545.045,Z 287.592,A -85,B 0,C 180,E1 -3471.865,E2 -3471.865} C_VEL
LIN {X 0,Y 545.032,Z 287.592,A -85,B 0,C 180,E1 -3474.531,E2 -3474.531} C_VEL
LIN {X 0,Y 545.069,Z 287.582,A -85,B 0,C 180,E1 -3477.211,E2 -3477.211} C_VEL
LIN {X 0,Y 545.063,Z 287.585,A -85,B 0,C 180,E1 -3479.81,E2 -3479.81} C_VEL
LIN {X 0,Y 545.058,Z 287.591,A -85,B 0,C 180,E1 -3482.342,E2 -3482.342} C_VEL
LIN {X 0,Y 545.045,Z 287.592,A -85,B 0,C 180,E1 -3484.816,E2 -3484.816} C_VEL
LIN {X 0,Y 545.032,Z 287.589,A -85,B 0,C 180,E1 -3487.241,E2 -3487.241} C_VEL
LIN {X 0,Y 545.117,Z 287.58,A -85,B 0,C 180,E1 -3490.414,E2 -3490.414} C_VEL
LIN {X 0,Y 545.054,Z 287.586,A -85,B 0,C 180,E1 -3493.52,E2 -3493.52} C_VEL
LIN {X 0,Y 545.084,Z 287.581,A -85,B 0,C 180,E1 -3495.819,E2 -3495.819} C_VEL
LIN {X 0,Y 545.112,Z 287.583,A -85,B 0,C 180,E1 -3498.849,E2 -3498.849} C_VEL
LIN {X 0,Y 545.093,Z 287.584,A -85,B 0,C 180,E1 -3501.846,E2 -3501.846} C_VEL
LIN {X 0,Y 545.161,Z 287.724,A -85,B 0,C 180,E1 -3503.941,E2 -3503.941} C_VEL
LIN {X 0,Y 545.599,Z 291.478,A -85,B 0,C 180,E1 -3504.641,E2 -3504.641} C_VEL
LIN {X 0,Y 545.348,Z 306.85,A -85,B 0,C 180,E1 -3507.414,E2 -3507.414} C_VEL
LIN {X 0,Y 545.256,Z 318.513,A -85,B 0,C 180,E1 -3509.503,E2 -3509.503} C_VEL
LIN {X 0,Y 546.569,Z 327.136,A -85,B 0,C 180,E1 -3509.654,E2 -3509.654} C_VEL
LIN {X 0,Y 546.225,Z 425.325,A -85,B 0,C 180,E1 -3510.967,E2 -3510.967} C_VEL
LIN {X 0,Y 546.052,Z 437.636,A -85,B 0,C 180,E1 -3511.267,E2 -3511.267} C_VEL
LIN {X 0,Y 545.857,Z 450.926,A -85,B 0,C 180,E1 -3511.752,E2 -3511.752} C_VEL
LIN {X 0,Y 545.678,Z 462.109,A -85,B 0,C 180,E1 -3512.306,E2 -3512.306} C_VEL
LIN {X 0,Y 545.468,Z 473.653,A -85,B 0,C 180,E1 -3513.046,E2 -3513.046} C_VEL
LIN {X 0,Y 545.284,Z 484.043,A -85,B 0,C 180,E1 -3513.879,E2 -3513.879} C_VEL
LIN {X 0,Y 545.105,Z 493.452,A -85,B 0,C 180,E1 -3514.807,E2 -3514.807} C_VEL
LIN {X 0,Y 544.903,Z 502.573,A -85,B 0,C 180,E1 -3515.922,E2 -3515.922} C_VEL
LIN {X 0,Y 544.809,Z 509.934,A -85,B 0,C 180,E1 -3517.039,E2 -3517.039} C_VEL
LIN {X 0,Y 544.712,Z 515.863,A -85,B 0,C 180,E1 -3518.158,E2 -3518.158} C_VEL
LIN {X 0,Y 544.639,Z 520.556,A -85,B 0,C 180,E1 -3519.282,E2 -3519.282} C_VEL
LIN {X 0,Y 544.614,Z 524.139,A -85,B 0,C 180,E1 -3520.408,E2 -3520.408} C_VEL
LIN {X 0,Y 544.618,Z 526.164,A -85,B 0,C 180,E1 -3521.264,E2 -3521.264} C_VEL
LIN {X 0,Y 544.566,Z 528.299,A -85,B 0,C 180,E1 -3522.673,E2 -3522.673} C_VEL
LIN {X 0,Y 544.554,Z 528.864,A -85,B 0,C 180,E1 -3523.432,E2 -3523.432} C_VEL
LIN {X 0,Y 544.589,Z 528.895,A -85,B 0,C 180,E1 -3524.56,E2 -3524.56} C_VEL
LIN {X 0,Y 544.539,Z 527.964,A -85,B 0,C 180,E1 -3525.725,E2 -3525.725} C_VEL
LIN {X 0,Y 544.567,Z 526.812,A -85,B 0,C 180,E1 -3526.494,E2 -3526.494} C_VEL
LIN {X 0,Y 544.621,Z 524.222,A -85,B 0,C 180,E1 -3527.652,E2 -3527.652} C_VEL
LIN {X 0,Y 544.668,Z 520.518,A -85,B 0,C 180,E1 -3528.818,E2 -3528.818} C_VEL
LIN {X 0,Y 544.746,Z 514.711,A -85,B 0,C 180,E1 -3530.168,E2 -3530.168} C_VEL
LIN {X 0,Y 544.787,Z 509.202,A -85,B 0,C 180,E1 -3531.174,E2 -3531.174} C_VEL
LIN {X 0,Y 544.95,Z 501.166,A -85,B 0,C 180,E1 -3532.361,E2 -3532.361} C_VEL
LIN {X 0,Y 545.086,Z 492.759,A -85,B 0,C 180,E1 -3533.357,E2 -3533.357} C_VEL
LIN {X 0,Y 545.303,Z 482.389,A -85,B 0,C 180,E1 -3534.356,E2 -3534.356} C_VEL
LIN {X 0,Y 545.483,Z 472.053,A -85,B 0,C 180,E1 -3535.161,E2 -3535.161} C_VEL
LIN {X 0,Y 545.744,Z 460.918,A -85,B 0,C 180,E1 -3535.847,E2 -3535.847} C_VEL
LIN {X 0,Y 545.886,Z 448.956,A -85,B 0,C 180,E1 -3536.421,E2 -3536.421} C_VEL
LIN {X 0,Y 546.096,Z 435.711,A -85,B 0,C 180,E1 -3536.882,E2 -3536.882} C_VEL
LIN {X 0,Y 546.227,Z 422.961,A -85,B 0,C 180,E1 -3537.164,E2 -3537.164} C_VEL
LIN {X 0,Y 546.45,Z 325.541,A -85,B 0,C 180,E1 -3538.46,E2 -3538.46} C_VEL
LIN {X 0,Y 545.253,Z 318.191,A -85,B 0,C 180,E1 -3538.614,E2 -3538.614} C_VEL
LIN {X 0,Y 545.417,Z 300.587,A -85,B 0,C 180,E1 -3541.74,E2 -3541.74} C_VEL
LIN {X 0,Y 545.366,Z 289.684,A -85,B 0,C 180,E1 -3543.65,E2 -3543.65} C_VEL
LIN {X 0,Y 545.072,Z 287.59,A -85,B 0,C 180,E1 -3544.06,E2 -3544.06} C_VEL
LIN {X 0,Y 545.028,Z 287.593,A -85,B 0,C 180,E1 -3547.303,E2 -3547.303} C_VEL
LIN {X 0,Y 545.057,Z 287.586,A -85,B 0,C 180,E1 -3550.142,E2 -3550.142} C_VEL
LIN {X 0,Y 545.031,Z 287.593,A -85,B 0,C 180,E1 -3552.693,E2 -3552.693} C_VEL
LIN {X 0,Y 545.013,Z 287.599,A -85,B 0,C 180,E1 -3555.171,E2 -3555.171} C_VEL
LIN {X 0,Y 545.043,Z 287.587,A -85,B 0,C 180,E1 -3557.894,E2 -3557.894} C_VEL
LIN {X 0,Y 545.067,Z 287.587,A -85,B 0,C 180,E1 -3560.817,E2 -3560.817} C_VEL
LIN {X 0,Y 545.033,Z 287.593,A -85,B 0,C 180,E1 -3563.619,E2 -3563.619} C_VEL
LIN {X 0,Y 545.039,Z 287.582,A -85,B 0,C 180,E1 -3566.326,E2 -3566.326} C_VEL
LIN {X 0,Y 545.052,Z 287.587,A -85,B 0,C 180,E1 -3568.951,E2 -3568.951} C_VEL
LIN {X 0,Y 545.064,Z 287.592,A -85,B 0,C 180,E1 -3571.506,E2 -3571.506} C_VEL
LIN {X 0,Y 545.019,Z 287.588,A -85,B 0,C 180,E1 -3574.506,E2 -3574.506} C_VEL
LIN {X 0,Y 545.022,Z 287.591,A -85,B 0,C 180,E1 -3577.242,E2 -3577.242} C_VEL
LIN {X 0,Y 545.106,Z 287.58,A -85,B 0,C 180,E1 -3580.415,E2 -3580.415} C_VEL
LIN {X 0,Y 545.01,Z 287.593,A -85,B 0,C 180,E1 -3583.519,E2 -3583.519} C_VEL
LIN {X 0,Y 545.055,Z 287.591,A -85,B 0,C 180,E1 -3585.819,E2 -3585.819} C_VEL
LIN {X 0,Y 545.061,Z 287.584,A -85,B 0,C 180,E1 -3588.848,E2 -3588.848} C_VEL
LIN {X 0,Y 545.053,Z 287.587,A -85,B 0,C 180,E1 -3591.846,E2 -3591.846} C_VEL
LIN {X 0,Y 545.145,Z 287.575,A -85,B 0,C 180,E1 -3594.823,E2 -3594.823} C_VEL
LIN {X 0,Y 545.165,Z 287.57,A -85,B 0,C 180,E1 -3597.784,E2 -3597.784} C_VEL
LIN {X 0,Y 545.197,Z 287.571,A -85,B 0,C 180,E1 -3600.739,E2 -3600.739} C_VEL
LIN {X 0,Y 545.142,Z 287.576,A -85,B 0,C 180,E1 -3602.956,E2 -3602.956} C_VEL
LIN {X 0,Y 545.114,Z 287.578,A -85,B 0,C 180,E1 -3605.92,E2 -3605.92} C_VEL
LIN {X 0,Y 545.054,Z 287.584,A -85,B 0,C 180,E1 -3608.154,E2 -3608.154} C_VEL
LIN {X 0,Y 545.101,Z 287.582,A -85,B 0,C 180,E1 -3611.151,E2 -3611.151} C_VEL
LIN {X 0,Y 545.055,Z 287.583,A -85,B 0,C 180,E1 -3614.181,E2 -3614.181} C_VEL
LIN {X 0,Y 545.057,Z 287.585,A -85,B 0,C 180,E1 -3617.419,E2 -3617.419} C_VEL
LIN {X 0,Y 545.08,Z 287.582,A -85,B 0,C 180,E1 -3620.373,E2 -3620.373} C_VEL
LIN {X 0,Y 545.061,Z 287.587,A -85,B 0,C 180,E1 -3623.56,E2 -3623.56} C_VEL
LIN {X 0,Y 545.039,Z 287.587,A -85,B 0,C 180,E1 -3626.003,E2 -3626.003} C_VEL
LIN {X 0,Y 545.056,Z 287.585,A -85,B 0,C 180,E1 -3628.744,E2 -3628.744} C_VEL
LIN {X 0,Y 545.051,Z 287.59,A -85,B 0,C 180,E1 -3631.679,E2 -3631.679} C_VEL
LIN {X 0,Y 545.053,Z 287.585,A -85,B 0,C 180,E1 -3634.565,E2 -3634.565} C_VEL
LIN {X 0,Y 545.024,Z 287.594,A -85,B 0,C 180,E1 -3637.305,E2 -3637.305} C_VEL
LIN {X 0,Y 545.058,Z 287.588,A -85,B 0,C 180,E1 -3640.144,E2 -3640.144} C_VEL
LIN {X 0,Y 545.04,Z 287.585,A -85,B 0,C 180,E1 -3643.111,E2 -3643.111} C_VEL
LIN {X 0,Y 545.044,Z 287.591,A -85,B 0,C 180,E1 -3646.227,E2 -3646.227} C_VEL
LIN {X 0,Y 545.076,Z 287.583,A -85,B 0,C 180,E1 -3648.886,E2 -3648.886} C_VEL
LIN {X 0,Y 545.074,Z 287.584,A -85,B 0,C 180,E1 -3650.819,E2 -3650.819} C_VEL
LIN {X 0,Y 545.031,Z 287.592,A -85,B 0,C 180,E1 -3653.62,E2 -3653.62} C_VEL
LIN {X 0,Y 545.062,Z 287.592,A -85,B 0,C 180,E1 -3656.329,E2 -3656.329} C_VEL
LIN {X 0,Y 545.063,Z 287.586,A -85,B 0,C 180,E1 -3658.953,E2 -3658.953} C_VEL
LIN {X 0,Y 545.079,Z 287.584,A -85,B 0,C 180,E1 -3661.507,E2 -3661.507} C_VEL
LIN {X 0,Y 545.067,Z 287.59,A -85,B 0,C 180,E1 -3664,E2 -3664} C_VEL
LIN {X 0,Y 545.081,Z 287.65,A -85,B 0,C 180,E1 -3666.4,E2 -3666.4} C_VEL
LIN {X 0,Y 546.132,Z 294.256,A -85,B 0,C 180,E1 -3667.473,E2 -3667.473} C_VEL
LIN {X 0,Y 545.865,Z 311.611,A -85,B 0,C 180,E1 -3670.142,E2 -3670.142} C_VEL
LIN {X 0,Y 545.554,Z 330.169,A -85,B 0,C 180,E1 -3672.959,E2 -3672.959} C_VEL
LIN {X 0,Y 545.315,Z 346.704,A -85,B 0,C 180,E1 -3675.441,E2 -3675.441} C_VEL
LIN {X 0,Y 546.489,Z 354.27,A -85,B 0,C 180,E1 -3675.574,E2 -3675.574} C_VEL
LIN {X 0,Y 546.243,Z 454.869,A -85,B 0,C 180,E1 -3676.918,E2 -3676.918} C_VEL
LIN {X 0,Y 546.079,Z 468.151,A -85,B 0,C 180,E1 -3677.245,E2 -3677.245} C_VEL
LIN {X 0,Y 545.887,Z 480.323,A -85,B 0,C 180,E1 -3677.689,E2 -3677.689} C_VEL
LIN {X 0,Y 545.764,Z 491.231,A -85,B 0,C 180,E1 -3678.222,E2 -3678.222} C_VEL
LIN {X 0,Y 545.503,Z 502.911,A -85,B 0,C 180,E1 -3678.952,E2 -3678.952} C_VEL
LIN {X 0,Y 545.291,Z 513.544,A -85,B 0,C 180,E1 -3679.793,E2 -3679.793} C_VEL
LIN {X 0,Y 545.111,Z 523.12,A -85,B 0,C 180,E1 -3680.727,E2 -3680.727} C_VEL
LIN {X 0,Y 544.971,Z 530.966,A -85,B 0,C 180,E1 -3681.659,E2 -3681.659} C_VEL
LIN {X 0,Y 544.823,Z 538.625,A -85,B 0,C 180,E1 -3682.775,E2 -3682.775} C_VEL
LIN {X 0,Y 544.778,Z 545.683,A -85,B 0,C 180,E1 -3684.077,E2 -3684.077} C_VEL
LIN {X 0,Y 544.628,Z 550.376,A -85,B 0,C 180,E1 -3685.189,E2 -3685.189} C_VEL
LIN {X 0,Y 544.669,Z 553.96,A -85,B 0,C 180,E1 -3686.302,E2 -3686.302} C_VEL
LIN {X 0,Y 544.651,Z 555.808,A -85,B 0,C 180,E1 -3687.042,E2 -3687.042} C_VEL
LIN {X 0,Y 544.546,Z 558.183,A -85,B 0,C 180,E1 -3688.522,E2 -3688.522} C_VEL
LIN {X 0,Y 544.541,Z 559,A -85,B 0,C 180,E1 -3690.001,E2 -3690.001} C_VEL
LIN {X 0,Y 544.546,Z 558.183,A -85,B 0,C 180,E1 -3691.48,E2 -3691.48} C_VEL
LIN {X 0,Y 544.651,Z 555.809,A -85,B 0,C 180,E1 -3692.959,E2 -3692.959} C_VEL
LIN {X 0,Y 544.684,Z 552.893,A -85,B 0,C 180,E1 -3694.07,E2 -3694.07} C_VEL
LIN {X 0,Y 544.654,Z 548.946,A -85,B 0,C 180,E1 -3695.183,E2 -3695.183} C_VEL
LIN {X 0,Y 544.739,Z 543.592,A -85,B 0,C 180,E1 -3696.349,E2 -3696.349} C_VEL
LIN {X 0,Y 544.86,Z 536.231,A -85,B 0,C 180,E1 -3697.598,E2 -3697.598} C_VEL
LIN {X 0,Y 545.017,Z 527.987,A -85,B 0,C 180,E1 -3698.715,E2 -3698.715} C_VEL
LIN {X 0,Y 545.2,Z 519.534,A -85,B 0,C 180,E1 -3699.648,E2 -3699.648} C_VEL
LIN {X 0,Y 545.38,Z 509.083,A -85,B 0,C 180,E1 -3700.582,E2 -3700.582} C_VEL
LIN {X 0,Y 545.617,Z 497.549,A -85,B 0,C 180,E1 -3701.407,E2 -3701.407} C_VEL
LIN {X 0,Y 545.819,Z 487.351,A -85,B 0,C 180,E1 -3701.984,E2 -3701.984} C_VEL
LIN {X 0,Y 545.959,Z 475.675,A -85,B 0,C 180,E1 -3702.5,E2 -3702.5} C_VEL
LIN {X 0,Y 546.127,Z 462.222,A -85,B 0,C 180,E1 -3702.921,E2 -3702.921} C_VEL
LIN {X 0,Y 546.266,Z 448.919,A -85,B 0,C 180,E1 -3703.178,E2 -3703.178} C_VEL
LIN {X 0,Y 546.484,Z 354.132,A -85,B 0,C 180,E1 -3704.428,E2 -3704.428} C_VEL
LIN {X 0,Y 545.348,Z 346.586,A -85,B 0,C 180,E1 -3704.581,E2 -3704.581} C_VEL
LIN {X 0,Y 545.701,Z 323.875,A -85,B 0,C 180,E1 -3708.005,E2 -3708.005} C_VEL
LIN {X 0,Y 546.023,Z 303.487,A -85,B 0,C 180,E1 -3711.125,E2 -3711.125} C_VEL
LIN {X 0,Y 546.085,Z 293.306,A -85,B 0,C 180,E1 -3712.712,E2 -3712.712} C_VEL
LIN {X 0,Y 545.048,Z 287.596,A -85,B 0,C 180,E1 -3713.684,E2 -3713.684} C_VEL
LIN {X 0,Y 545.071,Z 287.589,A -85,B 0,C 180,E1 -3716.001,E2 -3716.001} C_VEL
LIN {X 0,Y 545.074,Z 287.582,A -85,B 0,C 180,E1 -3718.745,E2 -3718.745} C_VEL
LIN {X 0,Y 545.062,Z 287.59,A -85,B 0,C 180,E1 -3721.679,E2 -3721.679} C_VEL
LIN {X 0,Y 545.063,Z 287.585,A -85,B 0,C 180,E1 -3724.565,E2 -3724.565} C_VEL
LIN {X 0,Y 545.034,Z 287.587,A -85,B 0,C 180,E1 -3727.305,E2 -3727.305} C_VEL
LIN {X 0,Y 545.068,Z 287.592,A -85,B 0,C 180,E1 -3730.143,E2 -3730.143} C_VEL
LIN {X 0,Y 545.041,Z 287.59,A -85,B 0,C 180,E1 -3732.694,E2 -3732.694} C_VEL
LIN {X 0,Y 545.033,Z 287.587,A -85,B 0,C 180,E1 -3735.171,E2 -3735.171} C_VEL
LIN {X 0,Y 545.068,Z 287.584,A -85,B 0,C 180,E1 -3737.896,E2 -3737.896} C_VEL
LIN {X 0,Y 545.081,Z 287.588,A -85,B 0,C 180,E1 -3740.818,E2 -3740.818} C_VEL
LIN {X 0,Y 545.037,Z 287.586,A -85,B 0,C 180,E1 -3743.619,E2 -3743.619} C_VEL
LIN {X 0,Y 545.068,Z 287.585,A -85,B 0,C 180,E1 -3746.328,E2 -3746.328} C_VEL
LIN {X 0,Y 545.068,Z 287.593,A -85,B 0,C 180,E1 -3748.952,E2 -3748.952} C_VEL
LIN {X 0,Y 545.086,Z 287.583,A -85,B 0,C 180,E1 -3751.507,E2 -3751.507} C_VEL
LIN {X 0,Y 545.056,Z 287.584,A -85,B 0,C 180,E1 -3753.998,E2 -3753.998} C_VEL
LIN {X 0,Y 545.036,Z 287.597,A -85,B 0,C 180,E1 -3757.242,E2 -3757.242} C_VEL
LIN {X 0,Y 545.12,Z 287.576,A -85,B 0,C 180,E1 -3760.415,E2 -3760.415} C_VEL
LIN {X 0,Y 545.068,Z 287.593,A -85,B 0,C 180,E1 -3763.521,E2 -3763.521} C_VEL
LIN {X 0,Y 545.094,Z 287.585,A -85,B 0,C 180,E1 -3765.82,E2 -3765.82} C_VEL
LIN {X 0,Y 545.12,Z 287.576,A -85,B 0,C 180,E1 -3768.849,E2 -3768.849} C_VEL
LIN {X 0,Y 545.086,Z 287.59,A -85,B 0,C 180,E1 -3771.846,E2 -3771.846} C_VEL
LIN {X 0,Y 545.163,Z 287.578,A -85,B 0,C 180,E1 -3774.08,E2 -3774.08} C_VEL
LIN {X 0,Y 545.161,Z 287.571,A -85,B 0,C 180,E1 -3777.044,E2 -3777.044} C_VEL
LIN {X 0,Y 545.206,Z 287.574,A -85,B 0,C 180,E1 -3780,E2 -3780} C_VEL
LIN {X 0,Y 545.164,Z 287.571,A -85,B 0,C 180,E1 -3782.956,E2 -3782.956} C_VEL
LIN {X 0,Y 545.137,Z 287.577,A -85,B 0,C 180,E1 -3785.92,E2 -3785.92} C_VEL
LIN {X 0,Y 545.11,Z 287.581,A -85,B 0,C 180,E1 -3788.9,E2 -3788.9} C_VEL
LIN {X 0,Y 545.109,Z 287.578,A -85,B 0,C 180,E1 -3791.905,E2 -3791.905} C_VEL
LIN {X 0,Y 545.088,Z 287.586,A -85,B 0,C 180,E1 -3794.943,E2 -3794.943} C_VEL
LIN {X 0,Y 545.07,Z 287.583,A -85,B 0,C 180,E1 -3798.026,E2 -3798.026} C_VEL
LIN {X 0,Y 545.094,Z 287.582,A -85,B 0,C 180,E1 -3800.372,E2 -3800.372} C_VEL
LIN {X 0,Y 545.078,Z 287.583,A -85,B 0,C 180,E1 -3803.559,E2 -3803.559} C_VEL
LIN {X 0,Y 545.076,Z 287.581,A -85,B 0,C 180,E1 -3806.001,E2 -3806.001} C_VEL
LIN {X 0,Y 545.07,Z 287.585,A -85,B 0,C 180,E1 -3808.744,E2 -3808.744} C_VEL
LIN {X 0,Y 545.06,Z 287.588,A -85,B 0,C 180,E1 -3811.678,E2 -3811.678} C_VEL
LIN {X 0,Y 545.061,Z 287.583,A -85,B 0,C 180,E1 -3814.564,E2 -3814.564} C_VEL
LIN {X 0,Y 545.059,Z 287.586,A -85,B 0,C 180,E1 -3816.996,E2 -3816.996} C_VEL
LIN {X 0,Y 544.352,Z 287.681,A -85,B 0,C 180,E1 -3817.612,E2 -3817.612} C_VEL
LIN {X 0,Y 541.49,Z 288.039,A -85,B 0,C 180,E1 -3818.613,E2 -3818.613} C_VEL
LIN {X 0,Y 539.104,Z 288.333,A -85,B 0,C 180,E1 -3819.419,E2 -3819.419} C_VEL
LIN {X 0,Y 538.094,Z 288.456,A -85,B 0,C 180,E1 -3820.041,E2 -3820.041} C_VEL
LIN {X 0,Y 538.018,Z 288.462,A -85,B 0,C 180,E1 -3820.252,E2 -3820.252} C_VEL
LIN {X 0,Y 537.999,Z 288.463,A -85,B 0,C 180,E1 -3822.984,E2 -3822.984} C_VEL
LIN {X 0,Y 538.021,Z 288.47,A -85,B 0,C 180,E1 -3825.926,E2 -3825.926} C_VEL
LIN {X 0,Y 538.05,Z 288.457,A -85,B 0,C 180,E1 -3829.252,E2 -3829.252} C_VEL
LIN {X 0,Y 537.987,Z 288.475,A -85,B 0,C 180,E1 -3832.121,E2 -3832.121} C_VEL
LIN {X 0,Y 537.996,Z 288.464,A -85,B 0,C 180,E1 -3834.915,E2 -3834.915} C_VEL
LIN {X 0,Y 538.019,Z 288.461,A -85,B 0,C 180,E1 -3837.617,E2 -3837.617} C_VEL
LIN {X 0,Y 538.015,Z 288.468,A -85,B 0,C 180,E1 -3840.238,E2 -3840.238} C_VEL
LIN {X 0,Y 538.035,Z 288.464,A -85,B 0,C 180,E1 -3842.794,E2 -3842.794} C_VEL
LIN {X 0,Y 537.988,Z 288.465,A -85,B 0,C 180,E1 -3845.289,E2 -3845.289} C_VEL
LIN {X 0,Y 538.016,Z 288.462,A -85,B 0,C 180,E1 -3848.042,E2 -3848.042} C_VEL
LIN {X 0,Y 538.082,Z 288.454,A -85,B 0,C 180,E1 -3850.147,E2 -3850.147} C_VEL
LIN {X 0,Y 538.003,Z 288.467,A -85,B 0,C 180,E1 -3853.298,E2 -3853.298} C_VEL
LIN {X 0,Y 538.056,Z 288.457,A -85,B 0,C 180,E1 -3855.63,E2 -3855.63} C_VEL
LIN {X 0,Y 538.073,Z 288.457,A -85,B 0,C 180,E1 -3858.701,E2 -3858.701} C_VEL
LIN {X 0,Y 538.057,Z 288.462,A -85,B 0,C 180,E1 -3861.739,E2 -3861.739} C_VEL
LIN {X 0,Y 538.131,Z 288.552,A -85,B 0,C 180,E1 -3863.821,E2 -3863.821} C_VEL
LIN {X 0,Y 538.601,Z 292.533,A -85,B 0,C 180,E1 -3864.571,E2 -3864.571} C_VEL
LIN {X 0,Y 538.351,Z 306.897,A -85,B 0,C 180,E1 -3867.193,E2 -3867.193} C_VEL
LIN {X 0,Y 538.255,Z 318.682,A -85,B 0,C 180,E1 -3869.31,E2 -3869.31} C_VEL
LIN {X 0,Y 539.672,Z 327.085,A -85,B 0,C 180,E1 -3869.463,E2 -3869.463} C_VEL
LIN {X 0,Y 539.324,Z 425.292,A -85,B 0,C 180,E1 -3870.793,E2 -3870.793} C_VEL
LIN {X 0,Y 539.163,Z 437.659,A -85,B 0,C 180,E1 -3871.096,E2 -3871.096} C_VEL
LIN {X 0,Y 538.943,Z 451.001,A -85,B 0,C 180,E1 -3871.587,E2 -3871.587} C_VEL
LIN {X 0,Y 538.731,Z 462.224,A -85,B 0,C 180,E1 -3872.149,E2 -3872.149} C_VEL
LIN {X 0,Y 538.504,Z 473.785,A -85,B 0,C 180,E1 -3872.898,E2 -3872.898} C_VEL
LIN {X 0,Y 538.297,Z 484.187,A -85,B 0,C 180,E1 -3873.742,E2 -3873.742} C_VEL
LIN {X 0,Y 538.071,Z 493.609,A -85,B 0,C 180,E1 -3874.682,E2 -3874.682} C_VEL
LIN {X 0,Y 537.854,Z 502.7,A -85,B 0,C 180,E1 -3875.811,E2 -3875.811} C_VEL
LIN {X 0,Y 537.735,Z 510.033,A -85,B 0,C 180,E1 -3876.943,E2 -3876.943} C_VEL
LIN {X 0,Y 537.631,Z 516.797,A -85,B 0,C 180,E1 -3878.267,E2 -3878.267} C_VEL
LIN {X 0,Y 537.564,Z 521.269,A -85,B 0,C 180,E1 -3879.405,E2 -3879.405} C_VEL
LIN {X 0,Y 537.519,Z 524.667,A -85,B 0,C 180,E1 -3880.547,E2 -3880.547} C_VEL
LIN {X 0,Y 537.536,Z 526.351,A -85,B 0,C 180,E1 -3881.309,E2 -3881.309} C_VEL
LIN {X 0,Y 537.467,Z 527.636,A -85,B 0,C 180,E1 -3882.076,E2 -3882.076} C_VEL
LIN {X 0,Y 537.472,Z 528.508,A -85,B 0,C 180,E1 -3882.843,E2 -3882.843} C_VEL
LIN {X 0,Y 537.473,Z 528.929,A -85,B 0,C 180,E1 -3883.613,E2 -3883.613} C_VEL
LIN {X 0,Y 537.499,Z 528.893,A -85,B 0,C 180,E1 -3884.63,E2 -3884.63} C_VEL
LIN {X 0,Y 537.439,Z 527.748,A -85,B 0,C 180,E1 -3885.938,E2 -3885.938} C_VEL
LIN {X 0,Y 537.531,Z 525.095,A -85,B 0,C 180,E1 -3887.361,E2 -3887.361} C_VEL
LIN {X 0,Y 537.564,Z 521.286,A -85,B 0,C 180,E1 -3888.681,E2 -3888.681} C_VEL
LIN {X 0,Y 537.67,Z 516.611,A -85,B 0,C 180,E1 -3889.867,E2 -3889.867} C_VEL
LIN {X 0,Y 537.717,Z 510.525,A -85,B 0,C 180,E1 -3891.064,E2 -3891.064} C_VEL
LIN {X 0,Y 537.865,Z 502.791,A -85,B 0,C 180,E1 -3892.266,E2 -3892.266} C_VEL
LIN {X 0,Y 538.031,Z 494.792,A -85,B 0,C 180,E1 -3893.274,E2 -3893.274} C_VEL
LIN {X 0,Y 538.236,Z 485.359,A -85,B 0,C 180,E1 -3894.245,E2 -3894.245} C_VEL
LIN {X 0,Y 538.448,Z 475.064,A -85,B 0,C 180,E1 -3895.099,E2 -3895.099} C_VEL
LIN {X 0,Y 538.725,Z 464.203,A -85,B 0,C 180,E1 -3895.823,E2 -3895.823} C_VEL
LIN {X 0,Y 538.962,Z 451.693,A -85,B 0,C 180,E1 -3896.474,E2 -3896.474} C_VEL
LIN {X 0,Y 539.135,Z 439.161,A -85,B 0,C 180,E1 -3896.948,E2 -3896.948} C_VEL
LIN {X 0,Y 539.306,Z 426.406,A -85,B 0,C 180,E1 -3897.275,E2 -3897.275} C_VEL
LIN {X 0,Y 539.476,Z 379.9,A -85,B 0,C 180,E1 -3897.921,E2 -3897.921} C_VEL
LIN {X 0,Y 539.535,Z 326.12,A -85,B 0,C 180,E1 -3898.644,E2 -3898.644} C_VEL
LIN {X 0,Y 538.238,Z 318.289,A -85,B 0,C 180,E1 -3898.809,E2 -3898.809} C_VEL
LIN {X 0,Y 538.428,Z 299.671,A -85,B 0,C 180,E1 -3902.118,E2 -3902.118} C_VEL
LIN {X 0,Y 538.338,Z 290.62,A -85,B 0,C 180,E1 -3903.717,E2 -3903.717} C_VEL
LIN {X 0,Y 538.037,Z 288.467,A -85,B 0,C 180,E1 -3904.117,E2 -3904.117} C_VEL
LIN {X 0,Y 537.997,Z 288.471,A -85,B 0,C 180,E1 -3907.169,E2 -3907.169} C_VEL
LIN {X 0,Y 538.002,Z 288.465,A -85,B 0,C 180,E1 -3909.798,E2 -3909.798} C_VEL
LIN {X 0,Y 537.98,Z 288.473,A -85,B 0,C 180,E1 -3912.788,E2 -3912.788} C_VEL
LIN {X 0,Y 537.986,Z 288.475,A -85,B 0,C 180,E1 -3915.136,E2 -3915.136} C_VEL
LIN {X 0,Y 537.991,Z 288.465,A -85,B 0,C 180,E1 -3918.223,E2 -3918.223} C_VEL
LIN {X 0,Y 538.001,Z 288.472,A -85,B 0,C 180,E1 -3921.169,E2 -3921.169} C_VEL
LIN {X 0,Y 537.985,Z 288.466,A -85,B 0,C 180,E1 -3924.088,E2 -3924.088} C_VEL
LIN {X 0,Y 538.022,Z 288.457,A -85,B 0,C 180,E1 -3926.727,E2 -3926.727} C_VEL
LIN {X 0,Y 537.996,Z 288.473,A -85,B 0,C 180,E1 -3929.56,E2 -3929.56} C_VEL
LIN {X 0,Y 538,Z 288.468,A -85,B 0,C 180,E1 -3931.948,E2 -3931.948} C_VEL
LIN {X 0,Y 538,Z 288.463,A -85,B 0,C 180,E1 -3934.464,E2 -3934.464} C_VEL
LIN {X 0,Y 538,Z 288.464,A -85,B 0,C 180,E1 -3936.928,E2 -3936.928} C_VEL
LIN {X 0,Y 538.071,Z 288.459,A -85,B 0,C 180,E1 -3940.148,E2 -3940.148} C_VEL
LIN {X 0,Y 537.957,Z 288.469,A -85,B 0,C 180,E1 -3943.297,E2 -3943.297} C_VEL
LIN {X 0,Y 538.028,Z 288.464,A -85,B 0,C 180,E1 -3945.63,E2 -3945.63} C_VEL
LIN {X 0,Y 538.013,Z 288.463,A -85,B 0,C 180,E1 -3948.7,E2 -3948.7} C_VEL
LIN {X 0,Y 538.022,Z 288.461,A -85,B 0,C 180,E1 -3951.739,E2 -3951.739} C_VEL
LIN {X 0,Y 538.105,Z 288.452,A -85,B 0,C 180,E1 -3954.755,E2 -3954.755} C_VEL
LIN {X 0,Y 538.138,Z 288.445,A -85,B 0,C 180,E1 -3957.755,E2 -3957.755} C_VEL
LIN {X 0,Y 538.167,Z 288.446,A -85,B 0,C 180,E1 -3960.748,E2 -3960.748} C_VEL
LIN {X 0,Y 538.107,Z 288.452,A -85,B 0,C 180,E1 -3962.995,E2 -3962.995} C_VEL
LIN {X 0,Y 538.072,Z 288.456,A -85,B 0,C 180,E1 -3965.998,E2 -3965.998} C_VEL
LIN {X 0,Y 538.023,Z 288.46,A -85,B 0,C 180,E1 -3968.262,E2 -3968.262} C_VEL
LIN {X 0,Y 538.074,Z 288.453,A -85,B 0,C 180,E1 -3971.597,E2 -3971.597} C_VEL
LIN {X 0,Y 538.028,Z 288.465,A -85,B 0,C 180,E1 -3975.144,E2 -3975.144} C_VEL
LIN {X 0,Y 538,Z 288.461,A -85,B 0,C 180,E1 -3978.271,E2 -3978.271} C_VEL
LIN {X 0,Y 538.026,Z 288.463,A -85,B 0,C 180,E1 -3980.652,E2 -3980.652} C_VEL
LIN {X 0,Y 537.998,Z 288.463,A -85,B 0,C 180,E1 -3983.878,E2 -3983.878} C_VEL
LIN {X 0,Y 537.985,Z 288.465,A -85,B 0,C 180,E1 -3986.37,E2 -3986.37} C_VEL
LIN {X 0,Y 538.023,Z 288.464,A -85,B 0,C 180,E1 -3988.934,E2 -3988.934} C_VEL
LIN {X 0,Y 538.002,Z 288.465,A -85,B 0,C 180,E1 -3991.888,E2 -3991.888} C_VEL
LIN {X 0,Y 538.003,Z 288.463,A -85,B 0,C 180,E1 -3994.618,E2 -3994.618} C_VEL
LIN {X 0,Y 537.992,Z 288.468,A -85,B 0,C 180,E1 -3997.17,E2 -3997.17} C_VEL
LIN {X 0,Y 538.005,Z 288.471,A -85,B 0,C 180,E1 -3999.799,E2 -3999.799} C_VEL
LIN {X 0,Y 537.994,Z 288.461,A -85,B 0,C 180,E1 -4002.789,E2 -4002.789} C_VEL
LIN {X 0,Y 537.999,Z 288.465,A -85,B 0,C 180,E1 -4005.138,E2 -4005.138} C_VEL
LIN {X 0,Y 538.019,Z 288.468,A -85,B 0,C 180,E1 -4008.227,E2 -4008.227} C_VEL
LIN {X 0,Y 538.007,Z 288.464,A -85,B 0,C 180,E1 -4011.17,E2 -4011.17} C_VEL
LIN {X 0,Y 537.986,Z 288.475,A -85,B 0,C 180,E1 -4014.09,E2 -4014.09} C_VEL
LIN {X 0,Y 538.028,Z 288.463,A -85,B 0,C 180,E1 -4016.728,E2 -4016.728} C_VEL
LIN {X 0,Y 538.011,Z 288.465,A -85,B 0,C 180,E1 -4019.56,E2 -4019.56} C_VEL
LIN {X 0,Y 538.043,Z 288.466,A -85,B 0,C 180,E1 -4022.652,E2 -4022.652} C_VEL
LIN {X 0,Y 538,Z 288.473,A -85,B 0,C 180,E1 -4025.291,E2 -4025.291} C_VEL
LIN {X 0,Y 538.042,Z 288.626,A -85,B 0,C 180,E1 -4026.266,E2 -4026.266} C_VEL
LIN {X 0,Y 539.175,Z 295.676,A -85,B 0,C 180,E1 -4027.427,E2 -4027.427} C_VEL
LIN {X 0,Y 538.874,Z 313.351,A -85,B 0,C 180,E1 -4030.179,E2 -4030.179} C_VEL
LIN {X 0,Y 538.529,Z 331.23,A -85,B 0,C 180,E1 -4032.925,E2 -4032.925} C_VEL
LIN {X 0,Y 538.309,Z 346.586,A -85,B 0,C 180,E1 -4035.25,E2 -4035.25} C_VEL
LIN {X 0,Y 539.649,Z 355.747,A -85,B 0,C 180,E1 -4035.41,E2 -4035.41} C_VEL
LIN {X 0,Y 539.347,Z 454.625,A -85,B 0,C 180,E1 -4036.747,E2 -4036.747} C_VEL
LIN {X 0,Y 539.151,Z 467.92,A -85,B 0,C 180,E1 -4037.078,E2 -4037.078} C_VEL
LIN {X 0,Y 538.928,Z 481.222,A -85,B 0,C 180,E1 -4037.575,E2 -4037.575} C_VEL
LIN {X 0,Y 538.726,Z 492.954,A -85,B 0,C 180,E1 -4038.178,E2 -4038.178} C_VEL
LIN {X 0,Y 538.472,Z 505.291,A -85,B 0,C 180,E1 -4038.997,E2 -4038.997} C_VEL
LIN {X 0,Y 538.223,Z 515.491,A -85,B 0,C 180,E1 -4039.848,E2 -4039.848} C_VEL
LIN {X 0,Y 538.044,Z 524.671,A -85,B 0,C 180,E1 -4040.793,E2 -4040.793} C_VEL
LIN {X 0,Y 537.848,Z 533.614,A -85,B 0,C 180,E1 -4041.926,E2 -4041.926} C_VEL
LIN {X 0,Y 537.73,Z 540.812,A -85,B 0,C 180,E1 -4043.057,E2 -4043.057} C_VEL
LIN {X 0,Y 537.677,Z 547.365,A -85,B 0,C 180,E1 -4044.375,E2 -4044.375} C_VEL
LIN {X 0,Y 537.557,Z 551.679,A -85,B 0,C 180,E1 -4045.502,E2 -4045.502} C_VEL
LIN {X 0,Y 537.591,Z 553.96,A -85,B 0,C 180,E1 -4046.253,E2 -4046.253} C_VEL
LIN {X 0,Y 537.551,Z 555.808,A -85,B 0,C 180,E1 -4047.003,E2 -4047.003} C_VEL
LIN {X 0,Y 537.451,Z 558.182,A -85,B 0,C 180,E1 -4048.502,E2 -4048.502} C_VEL
LIN {X 0,Y 537.442,Z 559,A -85,B 0,C 180,E1 -4050.001,E2 -4050.001} C_VEL
LIN {X 0,Y 537.451,Z 558.182,A -85,B 0,C 180,E1 -4051.499,E2 -4051.499} C_VEL
LIN {X 0,Y 537.551,Z 555.809,A -85,B 0,C 180,E1 -4052.998,E2 -4052.998} C_VEL
LIN {X 0,Y 537.603,Z 552.893,A -85,B 0,C 180,E1 -4054.124,E2 -4054.124} C_VEL
LIN {X 0,Y 537.588,Z 548.945,A -85,B 0,C 180,E1 -4055.251,E2 -4055.251} C_VEL
LIN {X 0,Y 537.652,Z 544.06,A -85,B 0,C 180,E1 -4056.335,E2 -4056.335} C_VEL
LIN {X 0,Y 537.773,Z 537.404,A -85,B 0,C 180,E1 -4057.51,E2 -4057.51} C_VEL
LIN {X 0,Y 537.943,Z 529.376,A -85,B 0,C 180,E1 -4058.642,E2 -4058.642} C_VEL
LIN {X 0,Y 538.114,Z 521.194,A -85,B 0,C 180,E1 -4059.586,E2 -4059.586} C_VEL
LIN {X 0,Y 538.339,Z 511.217,A -85,B 0,C 180,E1 -4060.532,E2 -4060.532} C_VEL
LIN {X 0,Y 538.593,Z 501.375,A -85,B 0,C 180,E1 -4061.288,E2 -4061.288} C_VEL
LIN {X 0,Y 538.732,Z 490.289,A -85,B 0,C 180,E1 -4061.974,E2 -4061.974} C_VEL
LIN {X 0,Y 538.978,Z 477.805,A -85,B 0,C 180,E1 -4062.568,E2 -4062.568} C_VEL
LIN {X 0,Y 539.151,Z 464.742,A -85,B 0,C 180,E1 -4063.019,E2 -4063.019} C_VEL
LIN {X 0,Y 539.336,Z 451.701,A -85,B 0,C 180,E1 -4063.302,E2 -4063.302} C_VEL
LIN {X 0,Y 539.562,Z 354.492,A -85,B 0,C 180,E1 -4064.609,E2 -4064.609} C_VEL
LIN {X 0,Y 538.337,Z 346.546,A -85,B 0,C 180,E1 -4064.751,E2 -4064.751} C_VEL
LIN {X 0,Y 538.708,Z 324.721,A -85,B 0,C 180,E1 -4068.087,E2 -4068.087} C_VEL
LIN {X 0,Y 539.068,Z 304.589,A -85,B 0,C 180,E1 -4071.21,E2 -4071.21} C_VEL
LIN {X 0,Y 539.107,Z 294.406,A -85,B 0,C 180,E1 -4072.82,E2 -4072.82} C_VEL
LIN {X 0,Y 538.007,Z 288.471,A -85,B 0,C 180,E1 -4073.842,E2 -4073.842} C_VEL
LIN {X 0,Y 538.038,Z 288.461,A -85,B 0,C 180,E1 -4076.367,E2 -4076.367} C_VEL
LIN {X 0,Y 538.034,Z 288.46,A -85,B 0,C 180,E1 -4078.933,E2 -4078.933} C_VEL
LIN {X 0,Y 538.014,Z 288.472,A -85,B 0,C 180,E1 -4081.887,E2 -4081.887} C_VEL
LIN {X 0,Y 538.012,Z 288.463,A -85,B 0,C 180,E1 -4084.617,E2 -4084.617} C_VEL
LIN {X 0,Y 538.003,Z 288.462,A -85,B 0,C 180,E1 -4087.169,E2 -4087.169} C_VEL
LIN {X 0,Y 538.013,Z 288.465,A -85,B 0,C 180,E1 -4089.798,E2 -4089.798} C_VEL
LIN {X 0,Y 537.991,Z 288.467,A -85,B 0,C 180,E1 -4092.789,E2 -4092.789} C_VEL
LIN {X 0,Y 538.004,Z 288.463,A -85,B 0,C 180,E1 -4095.137,E2 -4095.137} C_VEL
LIN {X 0,Y 538.028,Z 288.465,A -85,B 0,C 180,E1 -4098.226,E2 -4098.226} C_VEL
LIN {X 0,Y 538.014,Z 288.463,A -85,B 0,C 180,E1 -4101.169,E2 -4101.169} C_VEL
LIN {X 0,Y 537.993,Z 288.465,A -85,B 0,C 180,E1 -4104.09,E2 -4104.09} C_VEL
LIN {X 0,Y 538.035,Z 288.467,A -85,B 0,C 180,E1 -4106.727,E2 -4106.727} C_VEL
LIN {X 0,Y 538.017,Z 288.462,A -85,B 0,C 180,E1 -4109.559,E2 -4109.559} C_VEL
LIN {X 0,Y 538.024,Z 288.46,A -85,B 0,C 180,E1 -4111.949,E2 -4111.949} C_VEL
LIN {X 0,Y 538.022,Z 288.461,A -85,B 0,C 180,E1 -4114.464,E2 -4114.464} C_VEL
LIN {X 0,Y 538.012,Z 288.467,A -85,B 0,C 180,E1 -4116.928,E2 -4116.928} C_VEL
LIN {X 0,Y 538.084,Z 288.453,A -85,B 0,C 180,E1 -4120.148,E2 -4120.148} C_VEL
LIN {X 0,Y 538.015,Z 288.468,A -85,B 0,C 180,E1 -4123.299,E2 -4123.299} C_VEL
LIN {X 0,Y 538.065,Z 288.464,A -85,B 0,C 180,E1 -4125.631,E2 -4125.631} C_VEL
LIN {X 0,Y 538.08,Z 288.453,A -85,B 0,C 180,E1 -4128.701,E2 -4128.701} C_VEL
LIN {X 0,Y 538.053,Z 288.466,A -85,B 0,C 180,E1 -4131.739,E2 -4131.739} C_VEL
LIN {X 0,Y 538.116,Z 288.457,A -85,B 0,C 180,E1 -4134.002,E2 -4134.002} C_VEL
LIN {X 0,Y 538.127,Z 288.447,A -85,B 0,C 180,E1 -4137.005,E2 -4137.005} C_VEL
LIN {X 0,Y 538.176,Z 288.45,A -85,B 0,C 180,E1 -4140,E2 -4140} C_VEL
LIN {X 0,Y 538.131,Z 288.447,A -85,B 0,C 180,E1 -4142.994,E2 -4142.994} C_VEL
LIN {X 0,Y 538.093,Z 288.456,A -85,B 0,C 180,E1 -4145.997,E2 -4145.997} C_VEL
LIN {X 0,Y 538.06,Z 288.457,A -85,B 0,C 180,E1 -4149.018,E2 -4149.018} C_VEL
LIN {X 0,Y 538.069,Z 288.457,A -85,B 0,C 180,E1 -4152.063,E2 -4152.063} C_VEL
LIN {X 0,Y 538.047,Z 288.46,A -85,B 0,C 180,E1 -4155.144,E2 -4155.144} C_VEL
LIN {X 0,Y 538.025,Z 288.462,A -85,B 0,C 180,E1 -4158.27,E2 -4158.27} C_VEL
LIN {X 0,Y 538.04,Z 288.464,A -85,B 0,C 180,E1 -4160.651,E2 -4160.651} C_VEL
LIN {X 0,Y 538.009,Z 288.462,A -85,B 0,C 180,E1 -4163.878,E2 -4163.878} C_VEL
LIN {X 0,Y 538.038,Z 288.459,A -85,B 0,C 180,E1 -4166.367,E2 -4166.367} C_VEL
LIN {X 0,Y 538.032,Z 288.464,A -85,B 0,C 180,E1 -4168.933,E2 -4168.933} C_VEL
LIN {X 0,Y 538.011,Z 288.464,A -85,B 0,C 180,E1 -4171.887,E2 -4171.887} C_VEL
LIN {X 0,Y 538.011,Z 288.462,A -85,B 0,C 180,E1 -4174.617,E2 -4174.617} C_VEL
LIN {X 0,Y 538.001,Z 288.467,A -85,B 0,C 180,E1 -4177.169,E2 -4177.169} C_VEL
LIN {X 0,Y 538.018,Z 288.462,A -85,B 0,C 180,E1 -4180.252,E2 -4180.252} C_VEL
LIN {X 0,Y 537.366,Z 288.543,A -85,B 0,C 180,E1 -4180.877,E2 -4180.877} C_VEL
LIN {X 0,Y 534.507,Z 288.905,A -85,B 0,C 180,E1 -4181.892,E2 -4181.892} C_VEL
LIN {X 0,Y 532.078,Z 289.211,A -85,B 0,C 180,E1 -4182.709,E2 -4182.709} C_VEL
LIN {X 0,Y 531.031,Z 289.338,A -85,B 0,C 180,E1 -4183.34,E2 -4183.34} C_VEL
LIN {X 0,Y 530.944,Z 289.347,A -85,B 0,C 180,E1 -4183.553,E2 -4183.553} C_VEL
LIN {X 0,Y 530.946,Z 289.343,A -85,B 0,C 180,E1 -4186.503,E2 -4186.503} C_VEL
LIN {X 0,Y 530.984,Z 289.337,A -85,B 0,C 180,E1 -4188.976,E2 -4188.976} C_VEL
LIN {X 0,Y 530.953,Z 289.343,A -85,B 0,C 180,E1 -4191.528,E2 -4191.528} C_VEL
LIN {X 0,Y 530.952,Z 289.348,A -85,B 0,C 180,E1 -4194.379,E2 -4194.379} C_VEL
LIN {X 0,Y 530.968,Z 289.339,A -85,B 0,C 180,E1 -4197.133,E2 -4197.133} C_VEL
LIN {X 0,Y 530.97,Z 289.34,A -85,B 0,C 180,E1 -4199.803,E2 -4199.803} C_VEL
LIN {X 0,Y 530.976,Z 289.348,A -85,B 0,C 180,E1 -4202.475,E2 -4202.475} C_VEL
LIN {X 0,Y 530.958,Z 289.345,A -85,B 0,C 180,E1 -4204.939,E2 -4204.939} C_VEL
LIN {X 0,Y 530.978,Z 289.338,A -85,B 0,C 180,E1 -4207.898,E2 -4207.898} C_VEL
LIN {X 0,Y 530.984,Z 289.345,A -85,B 0,C 180,E1 -4210.676,E2 -4210.676} C_VEL
LIN {X 0,Y 530.964,Z 289.347,A -85,B 0,C 180,E1 -4213.07,E2 -4213.07} C_VEL
LIN {X 0,Y 531.014,Z 289.337,A -85,B 0,C 180,E1 -4215.435,E2 -4215.435} C_VEL
LIN {X 0,Y 531.032,Z 289.333,A -85,B 0,C 180,E1 -4218.549,E2 -4218.549} C_VEL
LIN {X 0,Y 531.033,Z 289.339,A -85,B 0,C 180,E1 -4221.628,E2 -4221.628} C_VEL
LIN {X 0,Y 531.06,Z 289.426,A -85,B 0,C 180,E1 -4223.71,E2 -4223.71} C_VEL
LIN {X 0,Y 531.601,Z 293.572,A -85,B 0,C 180,E1 -4224.499,E2 -4224.499} C_VEL
LIN {X 0,Y 531.365,Z 308.006,A -85,B 0,C 180,E1 -4227.156,E2 -4227.156} C_VEL
LIN {X 0,Y 531.27,Z 318.851,A -85,B 0,C 180,E1 -4229.111,E2 -4229.111} C_VEL
LIN {X 0,Y 532.829,Z 328.667,A -85,B 0,C 180,E1 -4229.291,E2 -4229.291} C_VEL
LIN {X 0,Y 532.424,Z 425.257,A -85,B 0,C 180,E1 -4230.614,E2 -4230.614} C_VEL
LIN {X 0,Y 532.271,Z 437.69,A -85,B 0,C 180,E1 -4230.921,E2 -4230.921} C_VEL
LIN {X 0,Y 532.052,Z 449.963,A -85,B 0,C 180,E1 -4231.371,E2 -4231.371} C_VEL
LIN {X 0,Y 531.778,Z 462.343,A -85,B 0,C 180,E1 -4231.987,E2 -4231.987} C_VEL
LIN {X 0,Y 531.531,Z 473.922,A -85,B 0,C 180,E1 -4232.747,E2 -4232.747} C_VEL
LIN {X 0,Y 531.302,Z 484.335,A -85,B 0,C 180,E1 -4233.602,E2 -4233.602} C_VEL
LIN {X 0,Y 531.04,Z 493.771,A -85,B 0,C 180,E1 -4234.554,E2 -4234.554} C_VEL
LIN {X 0,Y 530.804,Z 502.87,A -85,B 0,C 180,E1 -4235.698,E2 -4235.698} C_VEL
LIN {X 0,Y 530.671,Z 510.206,A -85,B 0,C 180,E1 -4236.845,E2 -4236.845} C_VEL
LIN {X 0,Y 530.587,Z 516.109,A -85,B 0,C 180,E1 -4237.994,E2 -4237.994} C_VEL
LIN {X 0,Y 530.477,Z 520.787,A -85,B 0,C 180,E1 -4239.147,E2 -4239.147} C_VEL
LIN {X 0,Y 530.471,Z 524.353,A -85,B 0,C 180,E1 -4240.302,E2 -4240.302} C_VEL
LIN {X 0,Y 530.443,Z 526.908,A -85,B 0,C 180,E1 -4241.462,E2 -4241.462} C_VEL
LIN {X 0,Y 530.378,Z 528.098,A -85,B 0,C 180,E1 -4242.24,E2 -4242.24} C_VEL
LIN {X 0,Y 530.368,Z 528.831,A -85,B 0,C 180,E1 -4243.018,E2 -4243.018} C_VEL
LIN {X 0,Y 530.401,Z 529.166,A -85,B 0,C 180,E1 -4243.798,E2 -4243.798} C_VEL
LIN {X 0,Y 530.413,Z 529.061,A -85,B 0,C 180,E1 -4244.704,E2 -4244.704} C_VEL
LIN {X 0,Y 530.344,Z 527.662,A -85,B 0,C 180,E1 -4246.157,E2 -4246.157} C_VEL
LIN {X 0,Y 530.43,Z 525.186,A -85,B 0,C 180,E1 -4247.452,E2 -4247.452} C_VEL
LIN {X 0,Y 530.48,Z 522.145,A -85,B 0,C 180,E1 -4248.539,E2 -4248.539} C_VEL
LIN {X 0,Y 530.598,Z 517.093,A -85,B 0,C 180,E1 -4249.877,E2 -4249.877} C_VEL
LIN {X 0,Y 530.655,Z 510.742,A -85,B 0,C 180,E1 -4251.155,E2 -4251.155} C_VEL
LIN {X 0,Y 530.832,Z 502.751,A -85,B 0,C 180,E1 -4252.41,E2 -4252.41} C_VEL
LIN {X 0,Y 531.005,Z 495.016,A -85,B 0,C 180,E1 -4253.393,E2 -4253.393} C_VEL
LIN {X 0,Y 531.258,Z 485.139,A -85,B 0,C 180,E1 -4254.418,E2 -4254.418} C_VEL
LIN {X 0,Y 531.508,Z 473.921,A -85,B 0,C 180,E1 -4255.345,E2 -4255.345} C_VEL
LIN {X 0,Y 531.819,Z 462.778,A -85,B 0,C 180,E1 -4256.077,E2 -4256.077} C_VEL
LIN {X 0,Y 532.022,Z 450.737,A -85,B 0,C 180,E1 -4256.687,E2 -4256.687} C_VEL
LIN {X 0,Y 532.224,Z 437.389,A -85,B 0,C 180,E1 -4257.18,E2 -4257.18} C_VEL
LIN {X 0,Y 532.423,Z 424.608,A -85,B 0,C 180,E1 -4257.489,E2 -4257.489} C_VEL
LIN {X 0,Y 532.767,Z 327.523,A -85,B 0,C 180,E1 -4258.817,E2 -4258.817} C_VEL
LIN {X 0,Y 531.231,Z 318.423,A -85,B 0,C 180,E1 -4259.002,E2 -4259.002} C_VEL
LIN {X 0,Y 531.444,Z 300.621,A -85,B 0,C 180,E1 -4262.183,E2 -4262.183} C_VEL
LIN {X 0,Y 531.348,Z 291.831,A -85,B 0,C 180,E1 -4263.746,E2 -4263.746} C_VEL
LIN {X 0,Y 530.978,Z 289.347,A -85,B 0,C 180,E1 -4264.23,E2 -4264.23} C_VEL
LIN {X 0,Y 530.958,Z 289.345,A -85,B 0,C 180,E1 -4267.507,E2 -4267.507} C_VEL
LIN {X 0,Y 530.954,Z 289.345,A -85,B 0,C 180,E1 -4270.434,E2 -4270.434} C_VEL
LIN {X 0,Y 530.926,Z 289.352,A -85,B 0,C 180,E1 -4273.277,E2 -4273.277} C_VEL
LIN {X 0,Y 530.962,Z 289.343,A -85,B 0,C 180,E1 -4275.622,E2 -4275.622} C_VEL
LIN {X 0,Y 530.934,Z 289.35,A -85,B 0,C 180,E1 -4278.981,E2 -4278.981} C_VEL
LIN {X 0,Y 530.945,Z 289.348,A -85,B 0,C 180,E1 -4281.528,E2 -4281.528} C_VEL
LIN {X 0,Y 530.945,Z 289.343,A -85,B 0,C 180,E1 -4284.379,E2 -4284.379} C_VEL
LIN {X 0,Y 530.957,Z 289.341,A -85,B 0,C 180,E1 -4287.133,E2 -4287.133} C_VEL
LIN {X 0,Y 530.942,Z 289.347,A -85,B 0,C 180,E1 -4289.802,E2 -4289.802} C_VEL
LIN {X 0,Y 530.953,Z 289.342,A -85,B 0,C 180,E1 -4292.478,E2 -4292.478} C_VEL
LIN {X 0,Y 530.936,Z 289.343,A -85,B 0,C 180,E1 -4294.939,E2 -4294.939} C_VEL
LIN {X 0,Y 530.967,Z 289.347,A -85,B 0,C 180,E1 -4297.898,E2 -4297.898} C_VEL
LIN {X 0,Y 530.969,Z 289.339,A -85,B 0,C 180,E1 -4300.676,E2 -4300.676} C_VEL
LIN {X 0,Y 530.925,Z 289.344,A -85,B 0,C 180,E1 -4303.069,E2 -4303.069} C_VEL
LIN {X 0,Y 530.989,Z 289.339,A -85,B 0,C 180,E1 -4305.435,E2 -4305.435} C_VEL
LIN {X 0,Y 530.975,Z 289.342,A -85,B 0,C 180,E1 -4308.549,E2 -4308.549} C_VEL
LIN {X 0,Y 530.97,Z 289.338,A -85,B 0,C 180,E1 -4311.628,E2 -4311.628} C_VEL
LIN {X 0,Y 531.066,Z 289.33,A -85,B 0,C 180,E1 -4314.685,E2 -4314.685} C_VEL
LIN {X 0,Y 531.111,Z 289.32,A -85,B 0,C 180,E1 -4317.725,E2 -4317.725} C_VEL
LIN {X 0,Y 531.137,Z 289.322,A -85,B 0,C 180,E1 -4320.758,E2 -4320.758} C_VEL
LIN {X 0,Y 531.047,Z 289.331,A -85,B 0,C 180,E1 -4323.035,E2 -4323.035} C_VEL
LIN {X 0,Y 531.033,Z 289.333,A -85,B 0,C 180,E1 -4326.078,E2 -4326.078} C_VEL
LIN {X 0,Y 530.972,Z 289.34,A -85,B 0,C 180,E1 -4328.372,E2 -4328.372} C_VEL
LIN {X 0,Y 531.038,Z 289.329,A -85,B 0,C 180,E1 -4331.669,E2 -4331.669} C_VEL
LIN {X 0,Y 531.009,Z 289.343,A -85,B 0,C 180,E1 -4334.951,E2 -4334.951} C_VEL
LIN {X 0,Y 530.971,Z 289.336,A -85,B 0,C 180,E1 -4337.724,E2 -4337.724} C_VEL
LIN {X 0,Y 531.016,Z 289.333,A -85,B 0,C 180,E1 -4340.128,E2 -4340.128} C_VEL
LIN {X 0,Y 530.932,Z 289.344,A -85,B 0,C 180,E1 -4342.574,E2 -4342.574} C_VEL
LIN {X 0,Y 530.945,Z 289.349,A -85,B 0,C 180,E1 -4345.061,E2 -4345.061} C_VEL
LIN {X 0,Y 530.957,Z 289.344,A -85,B 0,C 180,E1 -4347.599,E2 -4347.599} C_VEL
LIN {X 0,Y 530.945,Z 289.343,A -85,B 0,C 180,E1 -4350.199,E2 -4350.199} C_VEL
LIN {X 0,Y 530.96,Z 289.342,A -85,B 0,C 180,E1 -4352.867,E2 -4352.867} C_VEL
LIN {X 0,Y 530.943,Z 289.35,A -85,B 0,C 180,E1 -4355.621,E2 -4355.621} C_VEL
LIN {X 0,Y 530.957,Z 289.34,A -85,B 0,C 180,E1 -4358.654,E2 -4358.654} C_VEL
LIN {X 0,Y 530.974,Z 289.345,A -85,B 0,C 180,E1 -4361.438,E2 -4361.438} C_VEL
LIN {X 0,Y 530.968,Z 289.34,A -85,B 0,C 180,E1 -4364.549,E2 -4364.549} C_VEL
LIN {X 0,Y 530.968,Z 289.349,A -85,B 0,C 180,E1 -4367.836,E2 -4367.836} C_VEL
LIN {X 0,Y 530.98,Z 289.341,A -85,B 0,C 180,E1 -4370.557,E2 -4370.557} C_VEL
LIN {X 0,Y 530.947,Z 289.344,A -85,B 0,C 180,E1 -4373.442,E2 -4373.442} C_VEL
LIN {X 0,Y 530.996,Z 289.342,A -85,B 0,C 180,E1 -4376.495,E2 -4376.495} C_VEL
LIN {X 0,Y 530.964,Z 289.342,A -85,B 0,C 180,E1 -4379.357,E2 -4379.357} C_VEL
LIN {X 0,Y 531.008,Z 289.344,A -85,B 0,C 180,E1 -4382.469,E2 -4382.469} C_VEL
LIN {X 0,Y 530.968,Z 289.352,A -85,B 0,C 180,E1 -4384.942,E2 -4384.942} C_VEL
LIN {X 0,Y 530.985,Z 289.44,A -85,B 0,C 180,E1 -4386.1,E2 -4386.1} C_VEL
LIN {X 0,Y 532.215,Z 296.471,A -85,B 0,C 180,E1 -4387.279,E2 -4387.279} C_VEL
LIN {X 0,Y 531.928,Z 313.134,A -85,B 0,C 180,E1 -4389.909,E2 -4389.909} C_VEL
LIN {X 0,Y 531.53,Z 332.296,A -85,B 0,C 180,E1 -4392.892,E2 -4392.892} C_VEL
LIN {X 0,Y 531.263,Z 346.265,A -85,B 0,C 180,E1 -4395.043,E2 -4395.043} C_VEL
LIN {X 0,Y 532.803,Z 356.787,A -85,B 0,C 180,E1 -4395.236,E2 -4395.236} C_VEL
LIN {X 0,Y 532.438,Z 454.381,A -85,B 0,C 180,E1 -4396.572,E2 -4396.572} C_VEL
LIN {X 0,Y 532.223,Z 467.688,A -85,B 0,C 180,E1 -4396.907,E2 -4396.907} C_VEL
LIN {X 0,Y 531.973,Z 480.998,A -85,B 0,C 180,E1 -4397.41,E2 -4397.41} C_VEL
LIN {X 0,Y 531.77,Z 492.582,A -85,B 0,C 180,E1 -4398.012,E2 -4398.012} C_VEL
LIN {X 0,Y 531.511,Z 503.78,A -85,B 0,C 180,E1 -4398.754,E2 -4398.754} C_VEL
LIN {X 0,Y 531.204,Z 514.232,A -85,B 0,C 180,E1 -4399.616,E2 -4399.616} C_VEL
LIN {X 0,Y 531.049,Z 522.781,A -85,B 0,C 180,E1 -4400.479,E2 -4400.479} C_VEL
LIN {X 0,Y 530.868,Z 530.666,A -85,B 0,C 180,E1 -4401.436,E2 -4401.436} C_VEL
LIN {X 0,Y 530.674,Z 538.366,A -85,B 0,C 180,E1 -4402.582,E2 -4402.582} C_VEL
LIN {X 0,Y 530.583,Z 545.465,A -85,B 0,C 180,E1 -4403.918,E2 -4403.918} C_VEL
LIN {X 0,Y 530.459,Z 550.185,A -85,B 0,C 180,E1 -4405.06,E2 -4405.06} C_VEL
LIN {X 0,Y 530.516,Z 553.795,A -85,B 0,C 180,E1 -4406.203,E2 -4406.203} C_VEL
LIN {X 0,Y 530.457,Z 555.654,A -85,B 0,C 180,E1 -4406.963,E2 -4406.963} C_VEL
LIN {X 0,Y 530.41,Z 557.048,A -85,B 0,C 180,E1 -4407.723,E2 -4407.723} C_VEL
LIN {X 0,Y 530.344,Z 558.65,A -85,B 0,C 180,E1 -4409.241,E2 -4409.241} C_VEL
LIN {X 0,Y 530.344,Z 558.866,A -85,B 0,C 180,E1 -4410.001,E2 -4410.001} C_VEL
LIN {X 0,Y 530.361,Z 558.043,A -85,B 0,C 180,E1 -4411.519,E2 -4411.519} C_VEL
LIN {X 0,Y 530.41,Z 557.05,A -85,B 0,C 180,E1 -4412.279,E2 -4412.279} C_VEL
LIN {X 0,Y 530.457,Z 555.657,A -85,B 0,C 180,E1 -4413.039,E2 -4413.039} C_VEL
LIN {X 0,Y 530.522,Z 552.724,A -85,B 0,C 180,E1 -4414.179,E2 -4414.179} C_VEL
LIN {X 0,Y 530.525,Z 548.752,A -85,B 0,C 180,E1 -4415.321,E2 -4415.321} C_VEL
LIN {X 0,Y 530.566,Z 543.201,A -85,B 0,C 180,E1 -4416.551,E2 -4416.551} C_VEL
LIN {X 0,Y 530.733,Z 535.966,A -85,B 0,C 180,E1 -4417.802,E2 -4417.802} C_VEL
LIN {X 0,Y 530.914,Z 527.681,A -85,B 0,C 180,E1 -4418.949,E2 -4418.949} C_VEL
LIN {X 0,Y 531.109,Z 519.189,A -85,B 0,C 180,E1 -4419.906,E2 -4419.906} C_VEL
LIN {X 0,Y 531.366,Z 508.694,A -85,B 0,C 180,E1 -4420.864,E2 -4420.864} C_VEL
LIN {X 0,Y 531.631,Z 497.926,A -85,B 0,C 180,E1 -4421.657,E2 -4421.657} C_VEL
LIN {X 0,Y 531.905,Z 486.928,A -85,B 0,C 180,E1 -4422.302,E2 -4422.302} C_VEL
LIN {X 0,Y 532.09,Z 475.239,A -85,B 0,C 180,E1 -4422.831,E2 -4422.831} C_VEL
LIN {X 0,Y 532.292,Z 461.769,A -85,B 0,C 180,E1 -4423.263,E2 -4423.263} C_VEL
LIN {X 0,Y 532.47,Z 448.419,A -85,B 0,C 180,E1 -4423.525,E2 -4423.525} C_VEL
LIN {X 0,Y 532.665,Z 355.128,A -85,B 0,C 180,E1 -4424.791,E2 -4424.791} C_VEL
LIN {X 0,Y 531.313,Z 346.314,A -85,B 0,C 180,E1 -4424.956,E2 -4424.956} C_VEL
LIN {X 0,Y 531.706,Z 324.696,A -85,B 0,C 180,E1 -4428.308,E2 -4428.308} C_VEL
LIN {X 0,Y 532.114,Z 305.686,A -85,B 0,C 180,E1 -4431.298,E2 -4431.298} C_VEL
LIN {X 0,Y 532.281,Z 296.774,A -85,B 0,C 180,E1 -4432.719,E2 -4432.719} C_VEL
LIN {X 0,Y 530.963,Z 289.347,A -85,B 0,C 180,E1 -4433.987,E2 -4433.987} C_VEL
LIN {X 0,Y 530.999,Z 289.337,A -85,B 0,C 180,E1 -4436.745,E2 -4436.745} C_VEL
LIN {X 0,Y 530.983,Z 289.341,A -85,B 0,C 180,E1 -4439.323,E2 -4439.323} C_VEL
LIN {X 0,Y 530.969,Z 289.345,A -85,B 0,C 180,E1 -4442.1,E2 -4442.1} C_VEL
LIN {X 0,Y 530.97,Z 289.339,A -85,B 0,C 180,E1 -4444.85,E2 -4444.85} C_VEL
LIN {X 0,Y 530.967,Z 289.341,A -85,B 0,C 180,E1 -4447.508,E2 -4447.508} C_VEL
LIN {X 0,Y 530.965,Z 289.346,A -85,B 0,C 180,E1 -4450.435,E2 -4450.435} C_VEL
LIN {X 0,Y 530.936,Z 289.343,A -85,B 0,C 180,E1 -4453.278,E2 -4453.278} C_VEL
LIN {X 0,Y 530.979,Z 289.338,A -85,B 0,C 180,E1 -4455.622,E2 -4455.622} C_VEL
LIN {X 0,Y 530.993,Z 289.346,A -85,B 0,C 180,E1 -4458.564,E2 -4458.564} C_VEL
LIN {X 0,Y 530.957,Z 289.34,A -85,B 0,C 180,E1 -4461.529,E2 -4461.529} C_VEL
LIN {X 0,Y 530.953,Z 289.345,A -85,B 0,C 180,E1 -4464.38,E2 -4464.38} C_VEL
LIN {X 0,Y 530.97,Z 289.344,A -85,B 0,C 180,E1 -4467.133,E2 -4467.133} C_VEL
LIN {X 0,Y 530.963,Z 289.34,A -85,B 0,C 180,E1 -4469.802,E2 -4469.802} C_VEL
LIN {X 0,Y 530.979,Z 289.339,A -85,B 0,C 180,E1 -4472.475,E2 -4472.475} C_VEL
LIN {X 0,Y 530.954,Z 289.347,A -85,B 0,C 180,E1 -4474.94,E2 -4474.94} C_VEL
LIN {X 0,Y 530.98,Z 289.339,A -85,B 0,C 180,E1 -4477.898,E2 -4477.898} C_VEL
LIN {X 0,Y 530.995,Z 289.337,A -85,B 0,C 180,E1 -4480.677,E2 -4480.677} C_VEL
LIN {X 0,Y 530.974,Z 289.342,A -85,B 0,C 180,E1 -4483.07,E2 -4483.07} C_VEL
LIN {X 0,Y 531.022,Z 289.341,A -85,B 0,C 180,E1 -4485.436,E2 -4485.436} C_VEL
LIN {X 0,Y 531.038,Z 289.33,A -85,B 0,C 180,E1 -4488.55,E2 -4488.55} C_VEL
LIN {X 0,Y 531.003,Z 289.342,A -85,B 0,C 180,E1 -4491.628,E2 -4491.628} C_VEL
LIN {X 0,Y 531.073,Z 289.336,A -85,B 0,C 180,E1 -4493.923,E2 -4493.923} C_VEL
LIN {X 0,Y 531.094,Z 289.323,A -85,B 0,C 180,E1 -4496.966,E2 -4496.966} C_VEL
LIN {X 0,Y 531.147,Z 289.325,A -85,B 0,C 180,E1 -4500,E2 -4500} C_VEL
LIN {X 0,Y 531.099,Z 289.323,A -85,B 0,C 180,E1 -4503.034,E2 -4503.034} C_VEL
LIN {X 0,Y 531.052,Z 289.334,A -85,B 0,C 180,E1 -4506.077,E2 -4506.077} C_VEL
LIN {X 0,Y 531.02,Z 289.333,A -85,B 0,C 180,E1 -4509.138,E2 -4509.138} C_VEL
LIN {X 0,Y 531.033,Z 289.335,A -85,B 0,C 180,E1 -4512.225,E2 -4512.225} C_VEL
LIN {X 0,Y 530.997,Z 289.337,A -85,B 0,C 180,E1 -4515.35,E2 -4515.35} C_VEL
LIN {X 0,Y 530.986,Z 289.342,A -85,B 0,C 180,E1 -4518.521,E2 -4518.521} C_VEL
LIN {X 0,Y 531.001,Z 289.345,A -85,B 0,C 180,E1 -4520.938,E2 -4520.938} C_VEL
LIN {X 0,Y 530.964,Z 289.34,A -85,B 0,C 180,E1 -4524.225,E2 -4524.225} C_VEL
LIN {X 0,Y 530.99,Z 289.34,A -85,B 0,C 180,E1 -4526.744,E2 -4526.744} C_VEL
LIN {X 0,Y 530.982,Z 289.346,A -85,B 0,C 180,E1 -4529.322,E2 -4529.322} C_VEL
LIN {X 0,Y 530.966,Z 289.34,A -85,B 0,C 180,E1 -4532.1,E2 -4532.1} C_VEL
LIN {X 0,Y 530.969,Z 289.34,A -85,B 0,C 180,E1 -4534.85,E2 -4534.85} C_VEL
LIN {X 0,Y 530.965,Z 289.349,A -85,B 0,C 180,E1 -4537.508,E2 -4537.508} C_VEL
LIN {X 0,Y 530.983,Z 289.338,A -85,B 0,C 180,E1 -4540.433,E2 -4540.433} C_VEL
LIN {X 0,Y 530.946,Z 289.347,A -85,B 0,C 180,E1 -4543.496,E2 -4543.496} C_VEL
LIN {X 0,Y 530.944,Z 289.347,A -85,B 0,C 180,E1 -4543.553,E2 -4543.553} C_VEL
LIN {X 0,Y 530.275,Z 289.43,A -85,B 0,C 180,E1 -4544.187,E2 -4544.187} C_VEL
LIN {X 0,Y 527.425,Z 289.782,A -85,B 0,C 180,E1 -4545.216,E2 -4545.216} C_VEL
LIN {X 0,Y 525.018,Z 290.087,A -85,B 0,C 180,E1 -4546.044,E2 -4546.044} C_VEL
LIN {X 0,Y 523.986,Z 290.21,A -85,B 0,C 180,E1 -4546.684,E2 -4546.684} C_VEL
LIN {X 0,Y 523.902,Z 290.219,A -85,B 0,C 180,E1 -4546.901,E2 -4546.901} C_VEL
LIN {X 0,Y 523.94,Z 290.222,A -85,B 0,C 180,E1 -4549.87,E2 -4549.87} C_VEL
LIN {X 0,Y 523.905,Z 290.22,A -85,B 0,C 180,E1 -4552.867,E2 -4552.867} C_VEL
LIN {X 0,Y 523.933,Z 290.217,A -85,B 0,C 180,E1 -4555.709,E2 -4555.709} C_VEL
LIN {X 0,Y 523.922,Z 290.225,A -85,B 0,C 180,E1 -4558.455,E2 -4558.455} C_VEL
LIN {X 0,Y 523.929,Z 290.217,A -85,B 0,C 180,E1 -4561.124,E2 -4561.124} C_VEL
LIN {X 0,Y 523.925,Z 290.218,A -85,B 0,C 180,E1 -4563.994,E2 -4563.994} C_VEL
LIN {X 0,Y 523.91,Z 290.222,A -85,B 0,C 180,E1 -4566.269,E2 -4566.269} C_VEL
LIN {X 0,Y 523.946,Z 290.224,A -85,B 0,C 180,E1 -4568.766,E2 -4568.766} C_VEL
LIN {X 0,Y 523.938,Z 290.219,A -85,B 0,C 180,E1 -4571.22,E2 -4571.22} C_VEL
LIN {X 0,Y 523.922,Z 290.218,A -85,B 0,C 180,E1 -4573.638,E2 -4573.638} C_VEL
LIN {X 0,Y 523.928,Z 290.216,A -85,B 0,C 180,E1 -4576.027,E2 -4576.027} C_VEL
LIN {X 0,Y 524.014,Z 290.206,A -85,B 0,C 180,E1 -4578.394,E2 -4578.394} C_VEL
LIN {X 0,Y 523.985,Z 290.218,A -85,B 0,C 180,E1 -4581.515,E2 -4581.515} C_VEL
LIN {X 0,Y 524.035,Z 290.355,A -85,B 0,C 180,E1 -4583.599,E2 -4583.599} C_VEL
LIN {X 0,Y 524.607,Z 294.647,A -85,B 0,C 180,E1 -4584.426,E2 -4584.426} C_VEL
LIN {X 0,Y 524.371,Z 309.147,A -85,B 0,C 180,E1 -4587.118,E2 -4587.118} C_VEL
LIN {X 0,Y 524.259,Z 319.086,A -85,B 0,C 180,E1 -4588.907,E2 -4588.907} C_VEL
LIN {X 0,Y 525.961,Z 328.581,A -85,B 0,C 180,E1 -4589.09,E2 -4589.09} C_VEL
LIN {X 0,Y 525.535,Z 426.336,A -85,B 0,C 180,E1 -4590.454,E2 -4590.454} C_VEL
LIN {X 0,Y 525.298,Z 439.275,A -85,B 0,C 180,E1 -4590.79,E2 -4590.79} C_VEL
LIN {X 0,Y 525.095,Z 452.259,A -85,B 0,C 180,E1 -4591.293,E2 -4591.293} C_VEL
LIN {X 0,Y 524.814,Z 464.033,A -85,B 0,C 180,E1 -4591.918,E2 -4591.918} C_VEL
LIN {X 0,Y 524.528,Z 475.334,A -85,B 0,C 180,E1 -4592.687,E2 -4592.687} C_VEL
LIN {X 0,Y 524.294,Z 485.538,A -85,B 0,C 180,E1 -4593.554,E2 -4593.554} C_VEL
LIN {X 0,Y 524.044,Z 493.924,A -85,B 0,C 180,E1 -4594.422,E2 -4594.422} C_VEL
LIN {X 0,Y 523.767,Z 503.036,A -85,B 0,C 180,E1 -4595.582,E2 -4595.582} C_VEL
LIN {X 0,Y 523.614,Z 509.954,A -85,B 0,C 180,E1 -4596.67,E2 -4596.67} C_VEL
LIN {X 0,Y 523.525,Z 515.382,A -85,B 0,C 180,E1 -4597.714,E2 -4597.714} C_VEL
LIN {X 0,Y 523.417,Z 520.252,A -85,B 0,C 180,E1 -4598.882,E2 -4598.882} C_VEL
LIN {X 0,Y 523.39,Z 524.002,A -85,B 0,C 180,E1 -4600.052,E2 -4600.052} C_VEL
LIN {X 0,Y 523.363,Z 527.047,A -85,B 0,C 180,E1 -4601.397,E2 -4601.397} C_VEL
LIN {X 0,Y 523.28,Z 528.496,A -85,B 0,C 180,E1 -4602.408,E2 -4602.408} C_VEL
LIN {X 0,Y 523.272,Z 529.148,A -85,B 0,C 180,E1 -4603.198,E2 -4603.198} C_VEL
LIN {X 0,Y 523.299,Z 529.405,A -85,B 0,C 180,E1 -4603.989,E2 -4603.989} C_VEL
LIN {X 0,Y 523.335,Z 529.216,A -85,B 0,C 180,E1 -4604.782,E2 -4604.782} C_VEL
LIN {X 0,Y 523.255,Z 528.601,A -85,B 0,C 180,E1 -4605.582,E2 -4605.582} C_VEL
LIN {X 0,Y 523.254,Z 527.576,A -85,B 0,C 180,E1 -4606.382,E2 -4606.382} C_VEL
LIN {X 0,Y 523.345,Z 525.266,A -85,B 0,C 180,E1 -4607.55,E2 -4607.55} C_VEL
LIN {X 0,Y 523.413,Z 521.708,A -85,B 0,C 180,E1 -4608.798,E2 -4608.798} C_VEL
LIN {X 0,Y 523.536,Z 517.105,A -85,B 0,C 180,E1 -4610.001,E2 -4610.001} C_VEL
LIN {X 0,Y 523.592,Z 510.96,A -85,B 0,C 180,E1 -4611.247,E2 -4611.247} C_VEL
LIN {X 0,Y 523.794,Z 503.073,A -85,B 0,C 180,E1 -4612.505,E2 -4612.505} C_VEL
LIN {X 0,Y 523.991,Z 495.242,A -85,B 0,C 180,E1 -4613.516,E2 -4613.516} C_VEL
LIN {X 0,Y 524.28,Z 485.377,A -85,B 0,C 180,E1 -4614.553,E2 -4614.553} C_VEL
LIN {X 0,Y 524.517,Z 475.551,A -85,B 0,C 180,E1 -4615.388,E2 -4615.388} C_VEL
LIN {X 0,Y 524.82,Z 464.86,A -85,B 0,C 180,E1 -4616.122,E2 -4616.122} C_VEL
LIN {X 0,Y 525.072,Z 453.329,A -85,B 0,C 180,E1 -4616.747,E2 -4616.747} C_VEL
LIN {X 0,Y 525.267,Z 441.787,A -85,B 0,C 180,E1 -4617.22,E2 -4617.22} C_VEL
LIN {X 0,Y 525.439,Z 428.69,A -85,B 0,C 180,E1 -4617.588,E2 -4617.588} C_VEL
LIN {X 0,Y 525.6,Z 410.503,A -85,B 0,C 180,E1 -4617.876,E2 -4617.876} C_VEL
LIN {X 0,Y 525.887,Z 328.243,A -85,B 0,C 180,E1 -4619.007,E2 -4619.007} C_VEL
LIN {X 0,Y 524.243,Z 318.567,A -85,B 0,C 180,E1 -4619.213,E2 -4619.213} C_VEL
LIN {X 0,Y 524.443,Z 300.71,A -85,B 0,C 180,E1 -4622.413,E2 -4622.413} C_VEL
LIN {X 0,Y 524.268,Z 292.043,A -85,B 0,C 180,E1 -4623.966,E2 -4623.966} C_VEL
LIN {X 0,Y 523.947,Z 290.223,A -85,B 0,C 180,E1 -4624.346,E2 -4624.346} C_VEL
LIN {X 0,Y 523.901,Z 290.223,A -85,B 0,C 180,E1 -4627.677,E2 -4627.677} C_VEL
LIN {X 0,Y 523.906,Z 290.221,A -85,B 0,C 180,E1 -4630.126,E2 -4630.126} C_VEL
LIN {X 0,Y 523.909,Z 290.222,A -85,B 0,C 180,E1 -4632.456,E2 -4632.456} C_VEL
LIN {X 0,Y 523.928,Z 290.224,A -85,B 0,C 180,E1 -4635.31,E2 -4635.31} C_VEL
LIN {X 0,Y 523.914,Z 290.221,A -85,B 0,C 180,E1 -4638.693,E2 -4638.693} C_VEL
LIN {X 0,Y 523.904,Z 290.221,A -85,B 0,C 180,E1 -4641.897,E2 -4641.897} C_VEL
LIN {X 0,Y 523.915,Z 290.222,A -85,B 0,C 180,E1 -4644.911,E2 -4644.911} C_VEL
LIN {X 0,Y 523.926,Z 290.224,A -85,B 0,C 180,E1 -4647.68,E2 -4647.68} C_VEL
LIN {X 0,Y 523.942,Z 290.214,A -85,B 0,C 180,E1 -4650.677,E2 -4650.677} C_VEL
LIN {X 0,Y 523.882,Z 290.229,A -85,B 0,C 180,E1 -4653.724,E2 -4653.724} C_VEL
LIN {X 0,Y 523.898,Z 290.222,A -85,B 0,C 180,E1 -4656.269,E2 -4656.269} C_VEL
LIN {X 0,Y 523.935,Z 290.215,A -85,B 0,C 180,E1 -4658.766,E2 -4658.766} C_VEL
LIN {X 0,Y 523.922,Z 290.218,A -85,B 0,C 180,E1 -4661.22,E2 -4661.22} C_VEL
LIN {X 0,Y 523.89,Z 290.224,A -85,B 0,C 180,E1 -4664.437,E2 -4664.437} C_VEL
LIN {X 0,Y 523.92,Z 290.215,A -85,B 0,C 180,E1 -4666.818,E2 -4666.818} C_VEL
LIN {X 0,Y 523.922,Z 290.217,A -85,B 0,C 180,E1 -4669.176,E2 -4669.176} C_VEL
LIN {X 0,Y 523.939,Z 290.222,A -85,B 0,C 180,E1 -4672.291,E2 -4672.291} C_VEL
LIN {X 0,Y 524.013,Z 290.21,A -85,B 0,C 180,E1 -4674.613,E2 -4674.613} C_VEL
LIN {X 0,Y 524.083,Z 290.195,A -85,B 0,C 180,E1 -4677.695,E2 -4677.695} C_VEL
LIN {X 0,Y 524.108,Z 290.197,A -85,B 0,C 180,E1 -4680.769,E2 -4680.769} C_VEL
LIN {X 0,Y 523.988,Z 290.21,A -85,B 0,C 180,E1 -4683.076,E2 -4683.076} C_VEL
LIN {X 0,Y 524,Z 290.21,A -85,B 0,C 180,E1 -4686.16,E2 -4686.16} C_VEL
LIN {X 0,Y 523.936,Z 290.218,A -85,B 0,C 180,E1 -4688.485,E2 -4688.485} C_VEL
LIN {X 0,Y 523.986,Z 290.208,A -85,B 0,C 180,E1 -4691.735,E2 -4691.735} C_VEL
LIN {X 0,Y 523.973,Z 290.218,A -85,B 0,C 180,E1 -4695.048,E2 -4695.048} C_VEL
LIN {X 0,Y 523.935,Z 290.212,A -85,B 0,C 180,E1 -4697.97,E2 -4697.97} C_VEL
LIN {X 0,Y 523.949,Z 290.214,A -85,B 0,C 180,E1 -4700.411,E2 -4700.411} C_VEL
LIN {X 0,Y 523.898,Z 290.225,A -85,B 0,C 180,E1 -4702.894,E2 -4702.894} C_VEL
LIN {X 0,Y 523.893,Z 290.227,A -85,B 0,C 180,E1 -4705.422,E2 -4705.422} C_VEL
LIN {X 0,Y 523.907,Z 290.219,A -85,B 0,C 180,E1 -4708.003,E2 -4708.003} C_VEL
LIN {X 0,Y 523.928,Z 290.219,A -85,B 0,C 180,E1 -4710.854,E2 -4710.854} C_VEL
LIN {X 0,Y 523.952,Z 290.219,A -85,B 0,C 180,E1 -4713.735,E2 -4713.735} C_VEL
LIN {X 0,Y 523.892,Z 290.221,A -85,B 0,C 180,E1 -4716.401,E2 -4716.401} C_VEL
LIN {X 0,Y 523.907,Z 290.22,A -85,B 0,C 180,E1 -4719.086,E2 -4719.086} C_VEL
LIN {X 0,Y 523.935,Z 290.216,A -85,B 0,C 180,E1 -4722.121,E2 -4722.121} C_VEL
LIN {X 0,Y 523.937,Z 290.218,A -85,B 0,C 180,E1 -4725.311,E2 -4725.311} C_VEL
LIN {X 0,Y 523.948,Z 290.216,A -85,B 0,C 180,E1 -4728.691,E2 -4728.691} C_VEL
LIN {X 0,Y 523.912,Z 290.22,A -85,B 0,C 180,E1 -4731.082,E2 -4731.082} C_VEL
LIN {X 0,Y 523.892,Z 290.228,A -85,B 0,C 180,E1 -4733.826,E2 -4733.826} C_VEL
LIN {X 0,Y 523.939,Z 290.219,A -85,B 0,C 180,E1 -4736.637,E2 -4736.637} C_VEL
LIN {X 0,Y 523.946,Z 290.217,A -85,B 0,C 180,E1 -4739.356,E2 -4739.356} C_VEL
LIN {X 0,Y 523.971,Z 290.22,A -85,B 0,C 180,E1 -4742.283,E2 -4742.283} C_VEL
LIN {X 0,Y 523.911,Z 290.23,A -85,B 0,C 180,E1 -4745.428,E2 -4745.428} C_VEL
LIN {X 0,Y 523.93,Z 290.349,A -85,B 0,C 180,E1 -4745.942,E2 -4745.942} C_VEL
LIN {X 0,Y 525.232,Z 297.53,A -85,B 0,C 180,E1 -4747.168,E2 -4747.168} C_VEL
LIN {X 0,Y 524.978,Z 312.908,A -85,B 0,C 180,E1 -4749.632,E2 -4749.632} C_VEL
LIN {X 0,Y 524.531,Z 332.086,A -85,B 0,C 180,E1 -4752.656,E2 -4752.656} C_VEL
LIN {X 0,Y 524.26,Z 346.072,A -85,B 0,C 180,E1 -4754.841,E2 -4754.841} C_VEL
LIN {X 0,Y 525.94,Z 357.294,A -85,B 0,C 180,E1 -4755.048,E2 -4755.048} C_VEL
